Yaskawa INFORM job: DEMO_ROOF_SIDE_0625_3PAINT_8.JBI

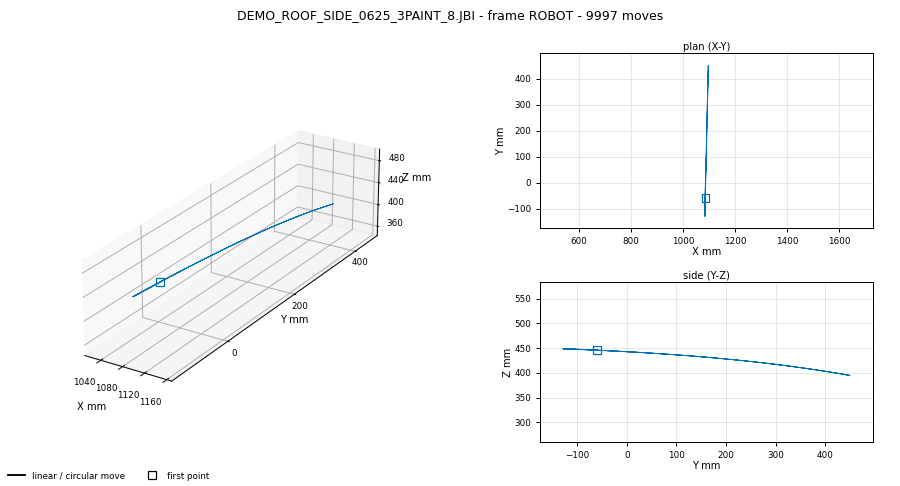
[picture p0: tool path of DEMO_ROOF_SIDE_0625_3PAINT_8.JBI in frame ROBOT, 9997 of 9997 moves have a stored position in this frame; points joined in program order, loops and branches not executed]
/JOB
//NAME DEMO_ROOF_SIDE_0625_3PAINT8
//POS
///NPOS 9997,0,0,0,0,0
///TOOL 0
///USER 0
///POSTYPE ROBOT
///RECTAN
///RCONF 1,0,0,0,0,0,0,0,0,0,0,0,0,0,0,0,0,0,0,0,0,0,0,0
C00000=1085.575,-60.075,446.143,174.285,17.982,152.948
C00001=1085.569,-60.325,446.155,174.283,17.980,152.948
C00002=1085.563,-60.574,446.167,174.282,17.979,152.948
C00003=1085.557,-60.824,446.178,174.280,17.978,152.948
C00004=1085.551,-61.074,446.189,174.279,17.976,152.948
C00005=1085.545,-61.323,446.201,174.277,17.974,152.948
C00006=1085.540,-61.573,446.212,174.276,17.973,152.948
C00007=1085.534,-61.823,446.223,174.274,17.972,152.948
C00008=1085.527,-62.072,446.235,174.273,17.970,152.948
C00009=1085.522,-62.322,446.246,174.272,17.969,152.948
C00010=1085.515,-62.572,446.257,174.270,17.968,152.948
C00011=1085.509,-62.821,446.269,174.269,17.966,152.948
C00012=1085.504,-63.071,446.281,174.267,17.965,152.948
C00013=1085.498,-63.321,446.292,174.265,17.963,152.948
C00014=1085.491,-63.571,446.303,174.264,17.962,152.948
C00015=1085.485,-63.820,446.315,174.263,17.960,152.948
C00016=1085.480,-64.069,446.325,174.261,17.959,152.948
C00017=1085.473,-64.320,446.337,174.260,17.958,152.948
C00018=1085.468,-64.569,446.349,174.258,17.956,152.948
C00019=1085.461,-64.842,446.360,174.257,17.955,152.948
C00020=1085.455,-65.116,446.373,174.254,17.953,152.948
C00021=1085.448,-65.389,446.385,174.253,17.951,152.948
C00022=1085.442,-65.662,446.398,174.252,17.950,152.948
C00023=1085.436,-65.912,446.409,174.250,17.948,152.948
C00024=1085.430,-66.162,446.420,174.248,17.947,152.948
C00025=1085.424,-66.411,446.431,174.247,17.946,152.948
C00026=1085.418,-66.661,446.443,174.246,17.944,152.948
C00027=1085.412,-66.911,446.454,174.244,17.943,152.948
C00028=1085.407,-67.160,446.465,174.243,17.942,152.948
C00029=1085.400,-67.410,446.476,174.241,17.940,152.948
C00030=1085.394,-67.660,446.487,174.240,17.939,152.948
C00031=1085.389,-67.909,446.498,174.238,17.937,152.948
C00032=1085.382,-68.159,446.510,174.237,17.936,152.948
C00033=1085.376,-68.409,446.521,174.235,17.935,152.948
C00034=1085.371,-68.658,446.532,174.234,17.933,152.948
C00035=1085.365,-68.909,446.544,174.232,17.932,152.948
C00036=1085.359,-69.158,446.555,174.231,17.931,152.948
C00037=1085.354,-69.407,446.565,174.229,17.929,152.948
C00038=1085.347,-69.658,446.577,174.228,17.928,152.948
C00039=1085.341,-69.907,446.588,174.226,17.926,152.948
C00040=1085.336,-70.157,446.598,174.225,17.925,152.948
C00041=1085.329,-70.406,446.610,174.223,17.924,152.948
C00042=1085.323,-70.656,446.621,174.222,17.922,152.948
C00043=1085.318,-70.905,446.632,174.220,17.921,152.948
C00044=1085.311,-71.155,446.643,174.219,17.920,152.948
C00045=1085.306,-71.405,446.654,174.217,17.918,152.948
C00046=1085.300,-71.655,446.666,174.216,17.917,152.948
C00047=1085.294,-71.905,446.677,174.214,17.915,152.948
C00048=1085.288,-72.154,446.688,174.213,17.914,152.948
C00049=1085.283,-72.404,446.699,174.211,17.913,152.949
C00050=1085.277,-72.653,446.710,174.210,17.911,152.948
C00051=1085.271,-72.904,446.721,174.208,17.910,152.948
C00052=1085.265,-73.153,446.732,174.207,17.909,152.949
C00053=1085.259,-73.403,446.743,174.205,17.907,152.949
C00054=1085.253,-73.652,446.754,174.204,17.906,152.949
C00055=1085.247,-73.902,446.765,174.202,17.904,152.949
C00056=1085.241,-74.152,446.776,174.201,17.903,152.949
C00057=1085.236,-74.401,446.787,174.199,17.902,152.949
C00058=1085.229,-74.651,446.798,174.198,17.900,152.949
C00059=1085.223,-74.901,446.809,174.196,17.899,152.949
C00060=1085.218,-75.150,446.820,174.195,17.898,152.949
C00061=1085.211,-75.400,446.830,174.193,17.896,152.949
C00062=1085.205,-75.650,446.841,174.192,17.895,152.949
C00063=1085.199,-75.899,446.852,174.190,17.894,152.949
C00064=1085.193,-76.149,446.863,174.188,17.893,152.949
C00065=1085.187,-76.399,446.874,174.187,17.891,152.949
C00066=1085.181,-76.648,446.885,174.185,17.890,152.949
C00067=1085.176,-76.898,446.896,174.184,17.889,152.949
C00068=1085.169,-77.148,446.906,174.182,17.888,152.949
C00069=1085.163,-77.398,446.917,174.181,17.886,152.949
C00070=1085.157,-77.647,446.927,174.179,17.885,152.949
C00071=1085.152,-77.897,446.938,174.178,17.883,152.949
C00072=1085.145,-78.147,446.950,174.176,17.882,152.949
C00073=1085.140,-78.397,446.960,174.175,17.881,152.949
C00074=1085.133,-78.646,446.971,174.174,17.880,152.949
C00075=1085.127,-78.895,446.982,174.172,17.879,152.949
C00076=1085.121,-79.145,446.993,174.171,17.878,152.949
C00077=1085.115,-79.395,447.004,174.169,17.876,152.949
C00078=1085.110,-79.645,447.014,174.168,17.875,152.949
C00079=1085.104,-79.894,447.025,174.166,17.874,152.950
C00080=1085.097,-80.144,447.035,174.165,17.872,152.950
C00081=1085.091,-80.394,447.046,174.163,17.871,152.950
C00082=1085.086,-80.643,447.057,174.162,17.870,152.950
C00083=1085.079,-80.920,447.069,174.160,17.869,152.950
C00084=1085.072,-81.195,447.081,174.158,17.868,152.950
C00085=1085.065,-81.470,447.093,174.157,17.866,152.950
C00086=1085.059,-81.746,447.104,174.154,17.865,152.950
C00087=1085.052,-81.995,447.114,174.153,17.863,152.950
C00088=1085.046,-82.245,447.126,174.152,17.862,152.950
C00089=1085.040,-82.495,447.136,174.150,17.861,152.950
C00090=1085.034,-82.744,447.146,174.149,17.860,152.950
C00091=1085.028,-82.994,447.157,174.147,17.859,152.950
C00092=1085.022,-83.244,447.168,174.146,17.858,152.950
C00093=1085.015,-83.493,447.178,174.144,17.857,152.950
C00094=1085.010,-83.743,447.189,174.143,17.855,152.950
C00095=1085.003,-83.993,447.199,174.141,17.854,152.950
C00096=1084.997,-84.243,447.210,174.139,17.853,152.951
C00097=1084.991,-84.492,447.221,174.138,17.851,152.951
C00098=1084.985,-84.742,447.231,174.136,17.850,152.951
C00099=1084.979,-84.992,447.241,174.135,17.849,152.951
C00100=1084.972,-85.241,447.252,174.133,17.848,152.951
C00101=1084.967,-85.492,447.262,174.132,17.847,152.951
C00102=1084.961,-85.741,447.273,174.131,17.846,152.951
C00103=1084.955,-85.990,447.283,174.129,17.845,152.951
C00104=1084.949,-86.240,447.294,174.128,17.844,152.951
C00105=1084.943,-86.491,447.305,174.126,17.842,152.951
C00106=1084.936,-86.740,447.315,174.124,17.841,152.951
C00107=1084.931,-86.990,447.325,174.123,17.840,152.951
C00108=1084.924,-87.239,447.335,174.121,17.839,152.951
C00109=1084.919,-87.488,447.346,174.120,17.838,152.951
C00110=1084.912,-87.739,447.356,174.118,17.836,152.951
C00111=1084.906,-87.988,447.367,174.117,17.835,152.952
C00112=1084.900,-88.238,447.378,174.115,17.834,152.952
C00113=1084.894,-88.488,447.388,174.114,17.834,152.952
C00114=1084.889,-88.737,447.398,174.113,17.832,152.952
C00115=1084.882,-88.986,447.409,174.111,17.831,152.952
C00116=1084.876,-89.237,447.419,174.109,17.830,152.952
C00117=1084.870,-89.486,447.430,174.108,17.829,152.952
C00118=1084.864,-89.737,447.440,174.106,17.827,152.952
C00119=1084.858,-89.986,447.451,174.105,17.826,152.952
C00120=1084.852,-90.235,447.461,174.103,17.825,152.952
C00121=1084.847,-90.485,447.471,174.101,17.824,152.952
C00122=1084.840,-90.734,447.481,174.101,17.823,152.952
C00123=1084.834,-90.985,447.492,174.099,17.822,152.952
C00124=1084.828,-91.234,447.502,174.097,17.821,152.952
C00125=1084.822,-91.485,447.512,174.096,17.820,152.953
C00126=1084.816,-91.734,447.523,174.094,17.819,152.953
C00127=1084.810,-91.984,447.533,174.093,17.817,152.953
C00128=1084.804,-92.233,447.543,174.091,17.816,152.953
C00129=1084.798,-92.483,447.554,174.089,17.815,152.953
C00130=1084.793,-92.733,447.564,174.088,17.814,152.953
C00131=1084.786,-92.982,447.574,174.087,17.813,152.953
C00132=1084.780,-93.233,447.585,174.085,17.812,152.953
C00133=1084.774,-93.482,447.595,174.084,17.811,152.953
C00134=1084.768,-93.732,447.605,174.082,17.810,152.953
C00135=1084.762,-93.981,447.616,174.080,17.809,152.953
C00136=1084.756,-94.231,447.626,174.079,17.807,152.953
C00137=1084.750,-94.480,447.636,174.077,17.806,152.953
C00138=1084.744,-94.731,447.646,174.076,17.805,152.954
C00139=1084.738,-94.980,447.656,174.074,17.804,152.954
C00140=1084.732,-95.230,447.667,174.073,17.804,152.954
C00141=1084.726,-95.480,447.676,174.072,17.803,152.954
C00142=1084.720,-95.729,447.687,174.070,17.801,152.954
C00143=1084.714,-95.979,447.697,174.068,17.800,152.954
C00144=1084.709,-96.228,447.708,174.067,17.799,152.954
C00145=1084.702,-96.478,447.717,174.065,17.798,152.954
C00146=1084.697,-96.728,447.727,174.063,17.797,152.954
C00147=1084.688,-97.066,447.741,174.062,17.796,152.954
C00148=1084.680,-97.404,447.755,174.060,17.794,152.954
C00149=1084.672,-97.741,447.769,174.058,17.793,152.954
C00150=1084.664,-98.079,447.782,174.055,17.791,152.955
C00151=1084.658,-98.328,447.793,174.054,17.790,152.955
C00152=1084.652,-98.578,447.802,174.053,17.789,152.955
C00153=1084.645,-98.828,447.812,174.051,17.788,152.955
C00154=1084.640,-99.077,447.823,174.050,17.787,152.955
C00155=1084.633,-99.328,447.833,174.048,17.786,152.955
C00156=1084.627,-99.577,447.842,174.046,17.785,152.955
C00157=1084.621,-99.827,447.853,174.045,17.784,152.955
C00158=1084.615,-100.077,447.863,174.044,17.784,152.955
C00159=1084.609,-100.326,447.872,174.042,17.783,152.956
C00160=1084.603,-100.576,447.883,174.040,17.782,152.956
C00161=1084.597,-100.826,447.893,174.039,17.781,152.956
C00162=1084.591,-101.076,447.902,174.037,17.779,152.956
C00163=1084.584,-101.325,447.912,174.035,17.778,152.956
C00164=1084.579,-101.575,447.923,174.035,17.778,152.956
C00165=1084.573,-101.825,447.932,174.033,17.777,152.956
C00166=1084.566,-102.074,447.942,174.031,17.776,152.956
C00167=1084.560,-102.324,447.952,174.030,17.775,152.956
C00168=1084.554,-102.574,447.962,174.028,17.774,152.957
C00169=1084.548,-102.824,447.972,174.026,17.773,152.957
C00170=1084.542,-103.073,447.982,174.026,17.772,152.957
C00171=1084.536,-103.323,447.992,174.024,17.771,152.957
C00172=1084.530,-103.573,448.002,174.022,17.770,152.957
C00173=1084.524,-103.822,448.011,174.021,17.769,152.957
C00174=1084.518,-104.072,448.022,174.019,17.768,152.957
C00175=1084.512,-104.322,448.032,174.017,17.767,152.957
C00176=1084.506,-104.571,448.041,174.016,17.766,152.957
C00177=1084.500,-104.821,448.051,174.015,17.765,152.957
C00178=1084.493,-105.070,448.061,174.013,17.764,152.958
C00179=1084.487,-105.320,448.071,174.011,17.763,152.958
C00180=1084.482,-105.570,448.081,174.010,17.762,152.958
C00181=1084.475,-105.820,448.090,174.009,17.762,152.958
C00182=1084.469,-106.070,448.100,174.007,17.761,152.958
C00183=1084.463,-106.319,448.110,174.006,17.760,152.958
C00184=1084.457,-106.569,448.120,174.004,17.758,152.958
C00185=1084.451,-106.819,448.130,174.002,17.758,152.958
C00186=1084.445,-107.069,448.140,174.000,17.757,152.959
C00187=1084.439,-107.319,448.149,173.999,17.756,152.959
C00188=1084.433,-107.568,448.159,173.998,17.755,152.959
C00189=1084.426,-107.818,448.169,173.996,17.754,152.959
C00190=1084.420,-108.067,448.179,173.994,17.753,152.959
C00191=1084.414,-108.317,448.188,173.993,17.752,152.959
C00192=1084.408,-108.567,448.198,173.992,17.752,152.959
C00193=1084.402,-108.817,448.208,173.990,17.751,152.959
C00194=1084.396,-109.067,448.217,173.988,17.750,152.960
C00195=1084.390,-109.317,448.227,173.987,17.749,152.960
C00196=1084.384,-109.567,448.237,173.985,17.748,152.960
C00197=1084.377,-109.816,448.247,173.984,17.747,152.960
C00198=1084.371,-110.065,448.256,173.983,17.746,152.960
C00199=1084.365,-110.315,448.266,173.981,17.746,152.960
C00200=1084.359,-110.565,448.276,173.979,17.745,152.960
C00201=1084.353,-110.815,448.285,173.978,17.744,152.960
C00202=1084.347,-111.064,448.294,173.976,17.743,152.961
C00203=1084.342,-111.284,448.303,173.975,17.742,152.961
C00204=1084.336,-111.504,448.312,173.974,17.742,152.961
C00205=1084.331,-111.724,448.320,173.972,17.741,152.961
C00206=1084.325,-111.944,448.329,173.970,17.740,152.961
C00207=1084.321,-112.163,448.337,173.970,17.740,152.961
C00208=1084.315,-112.383,448.346,173.968,17.739,152.961
C00209=1084.310,-112.604,448.354,173.967,17.738,152.961
C00210=1084.304,-112.823,448.362,173.965,17.737,152.962
C00211=1084.298,-113.096,448.373,173.963,17.736,152.962
C00212=1084.291,-113.370,448.384,173.962,17.735,152.962
C00213=1084.284,-113.643,448.394,173.960,17.734,152.962
C00214=1084.277,-113.917,448.405,173.958,17.734,152.962
C00215=1084.271,-114.167,448.414,173.957,17.733,152.962
C00216=1084.265,-114.417,448.424,173.956,17.732,152.962
C00217=1084.259,-114.667,448.433,173.954,17.731,152.963
C00218=1084.253,-114.916,448.443,173.952,17.731,152.963
C00219=1084.247,-115.166,448.452,173.951,17.730,152.963
C00220=1084.241,-115.416,448.461,173.950,17.729,152.963
C00221=1084.235,-115.666,448.471,173.948,17.729,152.963
C00222=1084.229,-115.916,448.480,173.946,17.727,152.963
C00223=1084.223,-116.165,448.490,173.945,17.727,152.963
C00224=1084.217,-116.415,448.499,173.943,17.726,152.964
C00225=1084.210,-116.665,448.509,173.942,17.725,152.964
C00226=1084.203,-116.914,448.518,173.940,17.724,152.964
C00227=1084.197,-117.164,448.527,173.939,17.724,152.964
C00228=1084.191,-117.414,448.537,173.937,17.723,152.964
C00229=1084.186,-117.663,448.546,173.936,17.722,152.964
C00230=1084.179,-117.913,448.556,173.934,17.721,152.964
C00231=1084.173,-118.163,448.565,173.933,17.721,152.965
C00232=1084.167,-118.412,448.575,173.931,17.720,152.965
C00233=1084.161,-118.663,448.584,173.929,17.720,152.965
C00234=1084.155,-118.913,448.593,173.927,17.719,152.965
C00235=1084.149,-119.163,448.603,173.927,17.718,152.965
C00236=1084.143,-119.412,448.612,173.925,17.718,152.965
C00237=1084.136,-119.661,448.621,173.923,17.716,152.966
C00238=1084.130,-119.911,448.631,173.921,17.715,152.966
C00239=1084.124,-120.161,448.640,173.920,17.715,152.966
C00240=1084.118,-120.410,448.650,173.919,17.714,152.966
C00241=1084.112,-120.661,448.659,173.917,17.714,152.966
C00242=1084.106,-120.911,448.668,173.915,17.713,152.966
C00243=1084.100,-121.160,448.677,173.914,17.712,152.966
C00244=1084.094,-121.410,448.687,173.912,17.712,152.967
C00245=1084.087,-121.659,448.696,173.911,17.711,152.967
C00246=1084.081,-121.910,448.705,173.910,17.711,152.967
C00247=1084.075,-122.159,448.714,173.908,17.710,152.967
C00248=1084.069,-122.409,448.724,173.906,17.709,152.967
C00249=1084.063,-122.658,448.733,173.904,17.708,152.968
C00250=1084.057,-122.908,448.743,173.903,17.708,152.968
C00251=1084.051,-123.158,448.751,173.901,17.707,152.968
C00252=1084.044,-123.408,448.760,173.900,17.706,152.968
C00253=1084.038,-123.658,448.770,173.899,17.706,152.968
C00254=1084.032,-123.907,448.780,173.897,17.705,152.968
C00255=1084.027,-124.157,448.789,173.895,17.704,152.969
C00256=1084.020,-124.407,448.797,173.893,17.703,152.969
C00257=1084.014,-124.656,448.807,173.892,17.703,152.969
C00258=1084.008,-124.906,448.816,173.891,17.702,152.969
C00259=1084.002,-125.157,448.825,173.889,17.702,152.969
C00260=1083.995,-125.405,448.834,173.888,17.701,152.969
C00261=1083.989,-125.655,448.843,173.886,17.701,152.970
C00262=1083.983,-125.905,448.853,173.884,17.700,152.970
C00263=1083.977,-126.156,448.862,173.882,17.699,152.970
C00264=1083.970,-126.405,448.871,173.882,17.699,152.970
C00265=1083.965,-126.654,448.880,173.880,17.698,152.970
C00266=1083.959,-126.905,448.889,173.878,17.697,152.970
C00267=1083.953,-127.154,448.898,173.877,17.697,152.971
C00268=1083.946,-127.404,448.907,173.875,17.696,152.971
C00269=1083.940,-127.654,448.917,173.873,17.695,152.971
C00270=1083.934,-127.903,448.925,173.872,17.695,152.971
C00271=1083.928,-128.160,448.935,173.871,17.694,152.971
C00272=1083.927,-128.416,448.946,173.869,17.692,152.971
C00273=1083.930,-128.671,448.958,173.869,17.689,152.971
C00274=1083.937,-128.924,448.972,173.869,17.684,152.970
C00275=1083.537,-128.945,448.838,173.825,17.800,153.000
C00276=1083.528,-128.693,448.824,173.825,17.805,153.001
C00277=1083.525,-128.438,448.812,173.826,17.808,153.001
C00278=1083.527,-128.182,448.801,173.827,17.810,153.001
C00279=1083.532,-127.926,448.791,173.828,17.811,153.001
C00280=1083.538,-127.676,448.782,173.829,17.812,153.001
C00281=1083.544,-127.426,448.773,173.831,17.812,153.001
C00282=1083.550,-127.176,448.763,173.833,17.813,153.001
C00283=1083.556,-126.927,448.755,173.835,17.814,153.001
C00284=1083.563,-126.677,448.745,173.836,17.814,153.001
C00285=1083.568,-126.427,448.736,173.838,17.815,153.000
C00286=1083.575,-126.177,448.727,173.839,17.816,153.000
C00287=1083.582,-125.927,448.718,173.840,17.816,153.000
C00288=1083.587,-125.678,448.709,173.842,17.817,153.000
C00289=1083.593,-125.428,448.700,173.844,17.817,153.000
C00290=1083.600,-125.178,448.691,173.846,17.819,152.999
C00291=1083.606,-124.929,448.681,173.847,17.819,152.999
C00292=1083.612,-124.678,448.672,173.848,17.820,152.999
C00293=1083.617,-124.429,448.663,173.850,17.820,152.999
C00294=1083.624,-124.180,448.654,173.851,17.821,152.999
C00295=1083.631,-123.930,448.645,173.853,17.821,152.999
C00296=1083.636,-123.679,448.636,173.855,17.822,152.998
C00297=1083.643,-123.430,448.626,173.857,17.823,152.998
C00298=1083.649,-123.180,448.617,173.858,17.823,152.998
C00299=1083.654,-122.931,448.607,173.859,17.824,152.998
C00300=1083.661,-122.681,448.599,173.861,17.825,152.998
C00301=1083.667,-122.431,448.590,173.862,17.825,152.998
C00302=1083.673,-122.181,448.580,173.864,17.826,152.997
C00303=1083.679,-121.931,448.571,173.866,17.827,152.997
C00304=1083.685,-121.682,448.561,173.867,17.828,152.997
C00305=1083.691,-121.432,448.552,173.868,17.828,152.997
C00306=1083.698,-121.182,448.543,173.870,17.829,152.997
C00307=1083.704,-120.932,448.534,173.872,17.829,152.997
C00308=1083.710,-120.683,448.524,173.874,17.830,152.996
C00309=1083.716,-120.433,448.515,173.874,17.831,152.996
C00310=1083.722,-120.183,448.505,173.876,17.832,152.996
C00311=1083.728,-119.933,448.497,173.878,17.833,152.996
C00312=1083.734,-119.684,448.487,173.880,17.834,152.996
C00313=1083.741,-119.434,448.478,173.881,17.834,152.996
C00314=1083.747,-119.184,448.469,173.882,17.835,152.996
C00315=1083.753,-118.934,448.459,173.884,17.836,152.995
C00316=1083.759,-118.685,448.449,173.886,17.836,152.995
C00317=1083.766,-118.435,448.440,173.887,17.837,152.995
C00318=1083.771,-118.186,448.431,173.889,17.838,152.995
C00319=1083.777,-117.935,448.422,173.891,17.838,152.995
C00320=1083.783,-117.686,448.412,173.892,17.839,152.995
C00321=1083.789,-117.436,448.403,173.893,17.840,152.995
C00322=1083.795,-117.186,448.393,173.895,17.840,152.994
C00323=1083.802,-116.936,448.384,173.897,17.841,152.994
C00324=1083.808,-116.686,448.374,173.898,17.842,152.994
C00325=1083.815,-116.437,448.365,173.899,17.842,152.994
C00326=1083.821,-116.187,448.355,173.901,17.844,152.994
C00327=1083.826,-115.938,448.346,173.903,17.845,152.994
C00328=1083.833,-115.688,448.337,173.904,17.846,152.993
C00329=1083.839,-115.438,448.327,173.905,17.846,152.993
C00330=1083.845,-115.189,448.318,173.907,17.847,152.993
C00331=1083.851,-114.939,448.308,173.909,17.848,152.993
C00332=1083.857,-114.689,448.298,173.910,17.849,152.993
C00333=1083.864,-114.439,448.289,173.912,17.849,152.993
C00334=1083.870,-114.189,448.279,173.913,17.850,152.993
C00335=1083.876,-113.940,448.270,173.915,17.851,152.992
C00336=1083.882,-113.666,448.260,173.917,17.852,152.992
C00337=1083.888,-113.392,448.249,173.918,17.853,152.992
C00338=1083.895,-113.118,448.238,173.920,17.853,152.992
C00339=1083.903,-112.844,448.228,173.922,17.854,152.992
C00340=1083.909,-112.595,448.218,173.924,17.856,152.992
C00341=1083.915,-112.345,448.209,173.924,17.856,152.992
C00342=1083.921,-112.095,448.199,173.926,17.857,152.992
C00343=1083.927,-111.846,448.190,173.928,17.858,152.991
C00344=1083.932,-111.596,448.180,173.930,17.859,152.991
C00345=1083.938,-111.346,448.170,173.931,17.860,152.991
C00346=1083.944,-111.096,448.161,173.932,17.860,152.991
C00347=1083.951,-110.846,448.151,173.934,17.861,152.991
C00348=1083.957,-110.597,448.141,173.935,17.862,152.991
C00349=1083.963,-110.347,448.132,173.937,17.863,152.990
C00350=1083.969,-110.097,448.122,173.939,17.864,152.990
C00351=1083.975,-109.847,448.113,173.940,17.864,152.990
C00352=1083.982,-109.597,448.103,173.942,17.865,152.990
C00353=1083.988,-109.348,448.094,173.943,17.866,152.990
C00354=1083.994,-109.098,448.083,173.945,17.868,152.990
C00355=1084.000,-108.849,448.074,173.947,17.869,152.990
C00356=1084.007,-108.599,448.064,173.948,17.869,152.990
C00357=1084.012,-108.349,448.054,173.949,17.870,152.990
C00358=1084.018,-108.099,448.044,173.951,17.871,152.989
C00359=1084.024,-107.849,448.035,173.953,17.872,152.989
C00360=1084.030,-107.599,448.025,173.954,17.873,152.989
C00361=1084.037,-107.350,448.015,173.955,17.873,152.989
C00362=1084.043,-107.100,448.005,173.957,17.874,152.989
C00363=1084.049,-106.850,447.996,173.958,17.875,152.989
C00364=1084.055,-106.600,447.986,173.960,17.876,152.989
C00365=1084.061,-106.351,447.976,173.962,17.877,152.989
C00366=1084.067,-106.101,447.967,173.963,17.878,152.989
C00367=1084.074,-105.852,447.956,173.964,17.879,152.988
C00368=1084.080,-105.602,447.947,173.966,17.880,152.988
C00369=1084.085,-105.352,447.937,173.968,17.881,152.988
C00370=1084.091,-105.102,447.927,173.969,17.882,152.988
C00371=1084.097,-104.852,447.917,173.971,17.883,152.988
C00372=1084.104,-104.603,447.907,173.972,17.883,152.988
C00373=1084.109,-104.353,447.897,173.974,17.884,152.988
C00374=1084.116,-104.103,447.887,173.975,17.885,152.988
C00375=1084.122,-103.853,447.878,173.977,17.886,152.987
C00376=1084.128,-103.604,447.868,173.979,17.887,152.987
C00377=1084.134,-103.354,447.857,173.980,17.888,152.987
C00378=1084.140,-103.104,447.848,173.981,17.889,152.987
C00379=1084.146,-102.854,447.838,173.983,17.890,152.987
C00380=1084.152,-102.605,447.828,173.984,17.892,152.987
C00381=1084.158,-102.355,447.818,173.986,17.893,152.987
C00382=1084.164,-102.105,447.808,173.988,17.894,152.987
C00383=1084.170,-101.855,447.799,173.989,17.895,152.987
C00384=1084.177,-101.606,447.788,173.990,17.895,152.987
C00385=1084.182,-101.356,447.778,173.992,17.896,152.987
C00386=1084.188,-101.106,447.769,173.993,17.897,152.986
C00387=1084.195,-100.857,447.758,173.995,17.898,152.986
C00388=1084.200,-100.607,447.748,173.997,17.899,152.986
C00389=1084.206,-100.357,447.739,173.998,17.900,152.986
C00390=1084.213,-100.108,447.728,173.999,17.901,152.986
C00391=1084.219,-99.858,447.719,174.001,17.902,152.986
C00392=1084.224,-99.608,447.709,174.003,17.903,152.986
C00393=1084.231,-99.359,447.698,174.004,17.904,152.986
C00394=1084.237,-99.109,447.689,174.006,17.905,152.986
C00395=1084.243,-98.859,447.679,174.008,17.906,152.985
C00396=1084.249,-98.610,447.668,174.009,17.907,152.985
C00397=1084.255,-98.360,447.659,174.010,17.908,152.985
C00398=1084.262,-98.110,447.648,174.012,17.909,152.985
C00399=1084.268,-97.860,447.638,174.013,17.910,152.985
C00400=1084.275,-97.582,447.627,174.015,17.911,152.985
C00401=1084.281,-97.304,447.616,174.017,17.912,152.985
C00402=1084.288,-97.026,447.605,174.018,17.913,152.985
C00403=1084.295,-96.748,447.593,174.020,17.914,152.985
C00404=1084.300,-96.498,447.583,174.021,17.916,152.985
C00405=1084.307,-96.249,447.572,174.023,17.917,152.985
C00406=1084.313,-95.999,447.563,174.025,17.918,152.985
C00407=1084.318,-95.750,447.552,174.026,17.919,152.984
C00408=1084.325,-95.500,447.542,174.028,17.920,152.984
C00409=1084.330,-95.250,447.532,174.029,17.922,152.984
C00410=1084.337,-95.001,447.522,174.031,17.923,152.984
C00411=1084.342,-94.751,447.512,174.032,17.923,152.984
C00412=1084.348,-94.501,447.502,174.034,17.924,152.984
C00413=1084.354,-94.251,447.491,174.035,17.926,152.984
C00414=1084.360,-94.002,447.481,174.037,17.927,152.984
C00415=1084.366,-93.752,447.471,174.038,17.928,152.984
C00416=1084.372,-93.503,447.460,174.040,17.929,152.984
C00417=1084.378,-93.253,447.450,174.042,17.930,152.984
C00418=1084.384,-93.003,447.439,174.043,17.932,152.984
C00419=1084.390,-92.753,447.430,174.044,17.932,152.984
C00420=1084.396,-92.503,447.419,174.045,17.933,152.984
C00421=1084.402,-92.253,447.409,174.047,17.934,152.983
C00422=1084.408,-92.004,447.398,174.049,17.936,152.983
C00423=1084.414,-91.754,447.389,174.050,17.937,152.983
C00424=1084.420,-91.505,447.378,174.052,17.938,152.983
C00425=1084.426,-91.255,447.368,174.054,17.939,152.983
C00426=1084.432,-91.005,447.357,174.055,17.941,152.983
C00427=1084.439,-90.756,447.347,174.057,17.942,152.983
C00428=1084.444,-90.505,447.337,174.058,17.943,152.983
C00429=1084.451,-90.256,447.326,174.059,17.944,152.983
C00430=1084.456,-90.006,447.316,174.061,17.945,152.983
C00431=1084.462,-89.757,447.305,174.062,17.946,152.983
C00432=1084.468,-89.507,447.295,174.064,17.947,152.983
C00433=1084.474,-89.257,447.285,174.065,17.948,152.983
C00434=1084.481,-89.007,447.274,174.067,17.949,152.983
C00435=1084.486,-88.757,447.264,174.069,17.951,152.982
C00436=1084.493,-88.508,447.254,174.070,17.952,152.982
C00437=1084.499,-88.259,447.243,174.072,17.953,152.982
C00438=1084.504,-88.009,447.233,174.073,17.954,152.982
C00439=1084.510,-87.759,447.222,174.074,17.955,152.982
C00440=1084.517,-87.509,447.211,174.076,17.956,152.982
C00441=1084.523,-87.259,447.202,174.077,17.957,152.982
C00442=1084.529,-87.010,447.191,174.079,17.959,152.982
C00443=1084.534,-86.760,447.180,174.080,17.960,152.982
C00444=1084.541,-86.511,447.170,174.082,17.961,152.982
C00445=1084.547,-86.260,447.159,174.084,17.962,152.982
C00446=1084.553,-86.011,447.149,174.085,17.964,152.982
C00447=1084.559,-85.761,447.139,174.087,17.965,152.982
C00448=1084.565,-85.512,447.128,174.088,17.966,152.982
C00449=1084.571,-85.262,447.117,174.090,17.967,152.982
C00450=1084.577,-85.012,447.107,174.091,17.968,152.982
C00451=1084.584,-84.762,447.097,174.092,17.969,152.982
C00452=1084.589,-84.513,447.086,174.094,17.970,152.982
C00453=1084.595,-84.264,447.075,174.095,17.971,152.981
C00454=1084.602,-84.013,447.065,174.097,17.973,152.981
C00455=1084.608,-83.764,447.054,174.098,17.974,152.981
C00456=1084.614,-83.514,447.044,174.100,17.975,152.981
C00457=1084.620,-83.265,447.033,174.102,17.977,152.981
C00458=1084.626,-83.014,447.022,174.103,17.978,152.981
C00459=1084.632,-82.765,447.012,174.105,17.979,152.981
C00460=1084.638,-82.515,447.001,174.106,17.980,152.981
C00461=1084.644,-82.266,446.990,174.108,17.981,152.981
C00462=1084.651,-82.016,446.980,174.109,17.983,152.981
C00463=1084.656,-81.766,446.970,174.111,17.984,152.981
C00464=1084.663,-81.491,446.958,174.113,17.985,152.981
C00465=1084.670,-81.215,446.946,174.114,17.987,152.981
C00466=1084.677,-80.939,446.934,174.116,17.988,152.981
C00467=1084.683,-80.663,446.923,174.117,17.989,152.981
C00468=1084.689,-80.414,446.912,174.119,17.990,152.981
C00469=1084.696,-80.164,446.901,174.120,17.991,152.981
C00470=1084.702,-79.915,446.890,174.122,17.993,152.981
C00471=1084.708,-79.665,446.879,174.124,17.994,152.980
C00472=1084.714,-79.415,446.868,174.125,17.995,152.980
C00473=1084.719,-79.165,446.858,174.127,17.996,152.980
C00474=1084.726,-78.916,446.848,174.128,17.998,152.980
C00475=1084.732,-78.666,446.837,174.130,17.999,152.980
C00476=1084.738,-78.416,446.826,174.131,18.001,152.980
C00477=1084.744,-78.166,446.815,174.133,18.002,152.980
C00478=1084.749,-77.917,446.804,174.134,18.003,152.980
C00479=1084.755,-77.667,446.793,174.136,18.004,152.980
C00480=1084.761,-77.417,446.782,174.137,18.006,152.980
C00481=1084.768,-77.168,446.772,174.139,18.007,152.980
C00482=1084.773,-76.918,446.761,174.140,18.008,152.980
C00483=1084.779,-76.668,446.750,174.142,18.010,152.980
C00484=1084.785,-76.418,446.739,174.143,18.011,152.980
C00485=1084.791,-76.169,446.728,174.145,18.013,152.980
C00486=1084.797,-75.919,446.717,174.146,18.014,152.980
C00487=1084.803,-75.669,446.706,174.147,18.015,152.980
C00488=1084.810,-75.420,446.696,174.149,18.016,152.980
C00489=1084.815,-75.170,446.685,174.150,18.017,152.980
C00490=1084.822,-74.920,446.674,174.152,18.018,152.980
C00491=1084.828,-74.671,446.663,174.153,18.020,152.980
C00492=1084.833,-74.421,446.652,174.155,18.021,152.980
C00493=1084.839,-74.172,446.641,174.156,18.023,152.980
C00494=1084.845,-73.922,446.630,174.158,18.024,152.980
C00495=1084.851,-73.672,446.619,174.159,18.025,152.980
C00496=1084.857,-73.423,446.608,174.161,18.027,152.980
C00497=1084.863,-73.172,446.597,174.162,18.028,152.980
C00498=1084.869,-72.923,446.586,174.164,18.029,152.980
C00499=1084.875,-72.673,446.575,174.165,18.031,152.980
C00500=1084.880,-72.424,446.564,174.167,18.032,152.980
C00501=1084.887,-72.174,446.553,174.168,18.033,152.980
C00502=1084.892,-71.924,446.542,174.170,18.035,152.980
C00503=1084.898,-71.675,446.531,174.171,18.036,152.980
C00504=1084.905,-71.425,446.520,174.173,18.038,152.980
C00505=1084.910,-71.175,446.509,174.174,18.039,152.980
C00506=1084.915,-70.925,446.498,174.176,18.040,152.980
C00507=1084.921,-70.676,446.486,174.177,18.042,152.980
C00508=1084.928,-70.426,446.475,174.179,18.043,152.980
C00509=1084.933,-70.177,446.464,174.180,18.044,152.979
C00510=1084.939,-69.927,446.453,174.182,18.046,152.980
C00511=1084.946,-69.677,446.442,174.183,18.048,152.980
C00512=1084.951,-69.428,446.431,174.184,18.049,152.980
C00513=1084.957,-69.178,446.420,174.186,18.050,152.979
C00514=1084.963,-68.928,446.409,174.188,18.052,152.980
C00515=1084.969,-68.678,446.398,174.189,18.053,152.980
C00516=1084.975,-68.430,446.386,174.191,18.054,152.979
C00517=1084.981,-68.179,446.375,174.192,18.056,152.979
C00518=1084.986,-67.930,446.364,174.193,18.057,152.980
C00519=1084.992,-67.680,446.353,174.195,18.059,152.979
C00520=1084.999,-67.430,446.342,174.197,18.060,152.979
C00521=1085.004,-67.180,446.331,174.198,18.062,152.979
C00522=1085.010,-66.932,446.319,174.199,18.063,152.980
C00523=1085.017,-66.681,446.308,174.201,18.064,152.979
C00524=1085.022,-66.432,446.297,174.202,18.066,152.979
C00525=1085.028,-66.181,446.285,174.204,18.067,152.979
C00526=1085.034,-65.932,446.274,174.205,18.068,152.979
C00527=1085.040,-65.683,446.263,174.207,18.070,152.979
C00528=1085.046,-65.409,446.250,174.209,18.072,152.979
C00529=1085.053,-65.135,446.238,174.211,18.074,152.979
C00530=1085.059,-64.861,446.226,174.212,18.075,152.979
C00531=1085.066,-64.588,446.214,174.214,18.076,152.979
C00532=1085.072,-64.339,446.202,174.215,18.078,152.979
C00533=1085.078,-64.089,446.191,174.216,18.079,152.979
C00534=1085.084,-63.839,446.180,174.218,18.081,152.979
C00535=1085.089,-63.590,446.169,174.219,18.082,152.979
C00536=1085.096,-63.340,446.157,174.221,18.084,152.979
C00537=1085.102,-63.091,446.146,174.222,18.085,152.979
C00538=1085.107,-62.840,446.134,174.225,18.087,152.979
C00539=1085.114,-62.591,446.123,174.226,18.088,152.979
C00540=1085.120,-62.341,446.111,174.228,18.090,152.979
C00541=1085.126,-62.092,446.100,174.229,18.091,152.979
C00542=1085.132,-61.843,446.089,174.230,18.093,152.979
C00543=1085.137,-61.592,446.077,174.232,18.094,152.979
C00544=1085.143,-61.343,446.066,174.233,18.096,152.979
C00545=1085.150,-61.093,446.054,174.235,18.097,152.979
C00546=1085.155,-60.844,446.043,174.236,18.099,152.979
C00547=1085.162,-60.594,446.032,174.238,18.100,152.979
C00548=1085.167,-60.344,446.020,174.239,18.101,152.979
C00549=1085.173,-60.094,446.009,174.241,18.103,152.979
C00550=1085.179,-59.845,445.998,174.242,18.104,152.979
C00551=1085.186,-59.595,445.986,174.244,18.105,152.979
C00552=1085.191,-59.346,445.975,174.245,18.107,152.979
C00553=1085.197,-59.096,445.962,174.247,18.109,152.979
C00554=1085.203,-58.846,445.951,174.248,18.110,152.979
C00555=1085.209,-58.596,445.940,174.249,18.112,152.979
C00556=1085.216,-58.347,445.929,174.251,18.113,152.979
C00557=1085.221,-58.097,445.917,174.253,18.114,152.979
C00558=1085.227,-57.848,445.905,174.254,18.116,152.979
C00559=1085.233,-57.598,445.894,174.255,18.117,152.979
C00560=1085.240,-57.349,445.882,174.257,18.119,152.980
C00561=1085.246,-57.099,445.871,174.259,18.120,152.979
C00562=1085.251,-56.849,445.860,174.261,18.122,152.979
C00563=1085.258,-56.599,445.848,174.262,18.124,152.979
C00564=1085.263,-56.350,445.837,174.264,18.125,152.979
C00565=1085.269,-56.100,445.824,174.265,18.127,152.980
C00566=1085.276,-55.850,445.813,174.267,18.128,152.979
C00567=1085.282,-55.601,445.801,174.268,18.129,152.979
C00568=1085.288,-55.351,445.790,174.269,18.131,152.979
C00569=1085.293,-55.101,445.778,174.271,18.132,152.980
C00570=1085.300,-54.851,445.767,174.272,18.134,152.980
C00571=1085.306,-54.602,445.755,174.274,18.135,152.979
C00572=1085.312,-54.352,445.744,174.275,18.137,152.979
C00573=1085.318,-54.102,445.731,174.277,18.138,152.980
C00574=1085.324,-53.853,445.720,174.278,18.140,152.980
C00575=1085.330,-53.603,445.709,174.280,18.141,152.980
C00576=1085.336,-53.354,445.696,174.281,18.142,152.979
C00577=1085.342,-53.104,445.685,174.283,18.144,152.979
C00578=1085.349,-52.854,445.673,174.285,18.146,152.980
C00579=1085.354,-52.605,445.662,174.286,18.148,152.980
C00580=1085.360,-52.355,445.650,174.288,18.149,152.980
C00581=1085.366,-52.106,445.638,174.289,18.151,152.980
C00582=1085.373,-51.856,445.627,174.291,18.152,152.980
C00583=1085.378,-51.606,445.614,174.292,18.153,152.980
C00584=1085.384,-51.356,445.603,174.294,18.155,152.980
C00585=1085.391,-51.107,445.591,174.295,18.156,152.980
C00586=1085.397,-50.857,445.579,174.296,18.158,152.980
C00587=1085.402,-50.607,445.568,174.298,18.160,152.980
C00588=1085.409,-50.358,445.556,174.299,18.161,152.980
C00589=1085.414,-50.108,445.545,174.301,18.162,152.980
C00590=1085.421,-49.859,445.533,174.303,18.164,152.980
C00591=1085.426,-49.609,445.520,174.304,18.166,152.980
C00592=1085.433,-49.336,445.508,174.306,18.167,152.980
C00593=1085.439,-49.065,445.494,174.307,18.169,152.980
C00594=1085.445,-48.792,445.482,174.310,18.171,152.980
C00595=1085.452,-48.520,445.468,174.311,18.173,152.980
C00596=1085.458,-48.271,445.457,174.312,18.174,152.980
C00597=1085.464,-48.021,445.445,174.314,18.176,152.980
C00598=1085.470,-47.772,445.433,174.315,18.177,152.980
C00599=1085.475,-47.521,445.421,174.317,18.179,152.980
C00600=1085.482,-47.272,445.409,174.318,18.180,152.980
C00601=1085.487,-47.023,445.397,174.319,18.182,152.980
C00602=1085.493,-46.773,445.384,174.321,18.183,152.980
C00603=1085.499,-46.523,445.374,174.323,18.186,152.980
C00604=1085.505,-46.273,445.361,174.324,18.187,152.980
C00605=1085.511,-46.024,445.349,174.326,18.189,152.980
C00606=1085.517,-45.775,445.337,174.327,18.190,152.980
C00607=1085.522,-45.524,445.325,174.329,18.192,152.980
C00608=1085.532,-45.122,445.306,174.331,18.194,152.980
C00609=1085.541,-44.720,445.286,174.334,18.197,152.980
C00610=1085.551,-44.318,445.267,174.336,18.200,152.980
C00611=1085.560,-43.916,445.247,174.339,18.203,152.980
C00612=1085.567,-43.666,445.235,174.340,18.204,152.981
C00613=1085.573,-43.416,445.223,174.341,18.206,152.981
C00614=1085.579,-43.167,445.212,174.343,18.207,152.981
C00615=1085.584,-42.917,445.199,174.344,18.209,152.981
C00616=1085.590,-42.667,445.187,174.346,18.210,152.981
C00617=1085.596,-42.418,445.175,174.347,18.212,152.981
C00618=1085.602,-42.168,445.163,174.348,18.214,152.981
C00619=1085.608,-41.918,445.150,174.351,18.216,152.981
C00620=1085.615,-41.669,445.138,174.352,18.217,152.981
C00621=1085.620,-41.419,445.127,174.353,18.219,152.981
C00622=1085.626,-41.169,445.114,174.355,18.220,152.981
C00623=1085.632,-40.920,445.102,174.356,18.222,152.981
C00624=1085.638,-40.670,445.090,174.358,18.223,152.981
C00625=1085.644,-40.420,445.077,174.359,18.225,152.981
C00626=1085.650,-40.171,445.066,174.361,18.227,152.981
C00627=1085.656,-39.922,445.053,174.363,18.229,152.981
C00628=1085.662,-39.672,445.041,174.364,18.230,152.981
C00629=1085.668,-39.422,445.029,174.366,18.232,152.981
C00630=1085.674,-39.172,445.016,174.367,18.233,152.981
C00631=1085.679,-38.923,445.004,174.368,18.235,152.981
C00632=1085.686,-38.674,444.992,174.370,18.236,152.981
C00633=1085.692,-38.424,444.980,174.371,18.238,152.981
C00634=1085.698,-38.173,444.968,174.373,18.240,152.981
C00635=1085.703,-37.924,444.956,174.375,18.242,152.981
C00636=1085.709,-37.674,444.943,174.376,18.243,152.981
C00637=1085.715,-37.425,444.931,174.378,18.245,152.981
C00638=1085.721,-37.175,444.919,174.379,18.246,152.981
C00639=1085.727,-36.926,444.906,174.381,18.248,152.981
C00640=1085.733,-36.676,444.894,174.382,18.249,152.981
C00641=1085.738,-36.426,444.882,174.383,18.251,152.982
C00642=1085.744,-36.177,444.869,174.385,18.254,152.982
C00643=1085.750,-35.927,444.857,174.387,18.255,152.982
C00644=1085.757,-35.678,444.844,174.388,18.257,152.982
C00645=1085.762,-35.429,444.832,174.390,18.258,152.982
C00646=1085.768,-35.179,444.819,174.391,18.260,152.982
C00647=1085.774,-34.929,444.806,174.392,18.261,152.982
C00648=1085.780,-34.679,444.794,174.394,18.263,152.982
C00649=1085.785,-34.430,444.782,174.396,18.265,152.982
C00650=1085.791,-34.180,444.769,174.397,18.267,152.982
C00651=1085.797,-33.930,444.757,174.399,18.269,152.982
C00652=1085.806,-33.561,444.739,174.401,18.271,152.982
C00653=1085.815,-33.193,444.720,174.403,18.273,152.982
C00654=1085.823,-32.824,444.702,174.405,18.275,152.982
C00655=1085.832,-32.455,444.683,174.408,18.278,152.982
C00656=1085.838,-32.205,444.671,174.409,18.280,152.982
C00657=1085.844,-31.956,444.659,174.411,18.282,152.982
C00658=1085.849,-31.706,444.646,174.412,18.283,152.982
C00659=1085.855,-31.456,444.633,174.413,18.285,152.983
C00660=1085.861,-31.206,444.621,174.415,18.287,152.983
C00661=1085.868,-30.957,444.608,174.417,18.289,152.983
C00662=1085.873,-30.708,444.595,174.418,18.290,152.983
C00663=1085.879,-30.458,444.583,174.420,18.292,152.983
C00664=1085.885,-30.208,444.570,174.421,18.294,152.983
C00665=1085.891,-29.958,444.558,174.423,18.295,152.983
C00666=1085.897,-29.709,444.544,174.424,18.297,152.983
C00667=1085.903,-29.459,444.532,174.426,18.299,152.983
C00668=1085.909,-29.210,444.520,174.427,18.301,152.983
C00669=1085.915,-28.960,444.508,174.429,18.302,152.983
C00670=1085.921,-28.711,444.494,174.430,18.304,152.983
C00671=1085.927,-28.461,444.482,174.432,18.305,152.983
C00672=1085.933,-28.211,444.469,174.433,18.307,152.983
C00673=1085.939,-27.961,444.457,174.435,18.309,152.983
C00674=1085.945,-27.712,444.444,174.437,18.311,152.983
C00675=1085.950,-27.463,444.431,174.438,18.312,152.983
C00676=1085.956,-27.213,444.419,174.440,18.314,152.983
C00677=1085.962,-26.963,444.406,174.441,18.316,152.983
C00678=1085.968,-26.714,444.393,174.442,18.317,152.984
C00679=1085.974,-26.464,444.380,174.444,18.319,152.984
C00680=1085.980,-26.214,444.368,174.446,18.321,152.984
C00681=1085.986,-25.965,444.355,174.447,18.323,152.984
C00682=1085.991,-25.715,444.342,174.448,18.325,152.984
C00683=1085.997,-25.466,444.329,174.450,18.326,152.984
C00684=1086.003,-25.216,444.316,174.452,18.328,152.984
C00685=1086.009,-24.966,444.303,174.453,18.330,152.984
C00686=1086.015,-24.717,444.291,174.455,18.331,152.984
C00687=1086.021,-24.467,444.278,174.456,18.333,152.984
C00688=1086.026,-24.218,444.265,174.457,18.335,152.984
C00689=1086.031,-23.968,444.252,174.459,18.337,152.984
C00690=1086.038,-23.719,444.239,174.461,18.339,152.984
C00691=1086.043,-23.469,444.226,174.463,18.340,152.984
C00692=1086.049,-23.219,444.214,174.464,18.342,152.984
C00693=1086.056,-22.970,444.201,174.465,18.344,152.984
C00694=1086.062,-22.720,444.188,174.467,18.345,152.984
C00695=1086.068,-22.470,444.175,174.469,18.347,152.984
C00696=1086.072,-22.221,444.162,174.470,18.349,152.985
C00697=1086.079,-21.972,444.149,174.471,18.351,152.985
C00698=1086.084,-21.722,444.136,174.473,18.353,152.985
C00699=1086.090,-21.472,444.124,174.474,18.354,152.985
C00700=1086.097,-21.223,444.110,174.476,18.356,152.985
C00701=1086.102,-20.972,444.097,174.478,18.358,152.985
C00702=1086.108,-20.723,444.084,174.479,18.360,152.985
C00703=1086.114,-20.473,444.071,174.480,18.361,152.985
C00704=1086.120,-20.224,444.058,174.482,18.363,152.985
C00705=1086.126,-19.974,444.046,174.484,18.365,152.985
C00706=1086.131,-19.725,444.032,174.485,18.367,152.985
C00707=1086.137,-19.475,444.019,174.487,18.369,152.985
C00708=1086.144,-19.225,444.006,174.488,18.370,152.985
C00709=1086.149,-18.976,443.994,174.489,18.372,152.985
C00710=1086.155,-18.727,443.980,174.492,18.374,152.985
C00711=1086.160,-18.477,443.967,174.493,18.375,152.985
C00712=1086.166,-18.228,443.954,174.494,18.377,152.986
C00713=1086.172,-17.978,443.941,174.496,18.379,152.986
C00714=1086.179,-17.728,443.928,174.497,18.381,152.986
C00715=1086.185,-17.479,443.915,174.499,18.383,152.986
C00716=1086.191,-17.206,443.901,174.501,18.384,152.986
C00717=1086.198,-16.933,443.886,174.502,18.386,152.986
C00718=1086.204,-16.660,443.872,174.504,18.388,152.986
C00719=1086.210,-16.388,443.858,174.506,18.390,152.986
C00720=1086.216,-16.138,443.844,174.508,18.392,152.986
C00721=1086.222,-15.889,443.832,174.509,18.394,152.986
C00722=1086.228,-15.639,443.818,174.510,18.396,152.986
C00723=1086.234,-15.390,443.805,174.512,18.397,152.986
C00724=1086.240,-15.140,443.792,174.513,18.399,152.986
C00725=1086.246,-14.891,443.779,174.515,18.401,152.986
C00726=1086.251,-14.640,443.766,174.517,18.403,152.986
C00727=1086.257,-14.391,443.752,174.518,18.404,152.986
C00728=1086.263,-14.142,443.739,174.520,18.406,152.987
C00729=1086.269,-13.892,443.726,174.521,18.408,152.987
C00730=1086.274,-13.642,443.712,174.523,18.410,152.987
C00731=1086.280,-13.393,443.699,174.524,18.412,152.987
C00732=1086.286,-13.143,443.686,174.526,18.413,152.987
C00733=1086.292,-12.893,443.672,174.527,18.415,152.987
C00734=1086.298,-12.644,443.659,174.529,18.417,152.987
C00735=1086.304,-12.395,443.645,174.531,18.419,152.987
C00736=1086.309,-12.145,443.633,174.532,18.420,152.987
C00737=1086.315,-11.895,443.619,174.533,18.422,152.987
C00738=1086.321,-11.646,443.606,174.535,18.425,152.987
C00739=1086.327,-11.396,443.593,174.537,18.426,152.987
C00740=1086.333,-11.146,443.579,174.538,18.428,152.987
C00741=1086.339,-10.897,443.566,174.539,18.430,152.988
C00742=1086.344,-10.648,443.552,174.541,18.431,152.988
C00743=1086.350,-10.398,443.539,174.543,18.433,152.988
C00744=1086.356,-10.148,443.526,174.544,18.435,152.988
C00745=1086.362,-9.899,443.512,174.546,18.437,152.988
C00746=1086.367,-9.649,443.498,174.547,18.438,152.988
C00747=1086.374,-9.400,443.485,174.549,18.441,152.988
C00748=1086.379,-9.150,443.472,174.550,18.443,152.988
C00749=1086.385,-8.901,443.459,174.552,18.444,152.988
C00750=1086.390,-8.651,443.445,174.553,18.446,152.988
C00751=1086.397,-8.402,443.432,174.556,18.448,152.988
C00752=1086.402,-8.152,443.418,174.557,18.450,152.988
C00753=1086.409,-7.902,443.404,174.558,18.451,152.988
C00754=1086.414,-7.652,443.391,174.560,18.453,152.988
C00755=1086.420,-7.403,443.378,174.562,18.455,152.988
C00756=1086.426,-7.153,443.364,174.563,18.457,152.989
C00757=1086.432,-6.904,443.351,174.564,18.459,152.989
C00758=1086.437,-6.654,443.337,174.566,18.460,152.989
C00759=1086.444,-6.405,443.323,174.567,18.462,152.989
C00760=1086.449,-6.155,443.310,174.569,18.464,152.989
C00761=1086.455,-5.906,443.296,174.571,18.466,152.989
C00762=1086.461,-5.655,443.283,174.572,18.467,152.989
C00763=1086.467,-5.406,443.270,174.573,18.469,152.989
C00764=1086.473,-5.156,443.256,174.576,18.471,152.989
C00765=1086.479,-4.907,443.242,174.577,18.473,152.989
C00766=1086.485,-4.658,443.229,174.578,18.475,152.989
C00767=1086.491,-4.408,443.215,174.580,18.476,152.989
C00768=1086.496,-4.159,443.201,174.582,18.478,152.989
C00769=1086.502,-3.909,443.188,174.583,18.480,152.989
C00770=1086.508,-3.659,443.174,174.585,18.482,152.989
C00771=1086.515,-3.410,443.161,174.586,18.483,152.990
C00772=1086.520,-3.160,443.147,174.588,18.485,152.989
C00773=1086.526,-2.911,443.133,174.589,18.488,152.990
C00774=1086.531,-2.661,443.119,174.591,18.489,152.990
C00775=1086.537,-2.412,443.106,174.593,18.491,152.990
C00776=1086.543,-2.162,443.092,174.594,18.493,152.990
C00777=1086.548,-1.913,443.078,174.596,18.495,152.990
C00778=1086.554,-1.663,443.064,174.597,18.496,152.990
C00779=1086.561,-1.413,443.051,174.599,18.499,152.990
C00780=1086.567,-1.140,443.035,174.601,18.500,152.990
C00781=1086.573,-0.865,443.020,174.603,18.503,152.990
C00782=1086.579,-0.591,443.005,174.604,18.505,152.990
C00783=1086.586,-0.316,442.990,174.606,18.507,152.991
C00784=1086.591,-0.067,442.976,174.607,18.509,152.991
C00785=1086.597,0.183,442.962,174.609,18.510,152.991
C00786=1086.602,0.432,442.948,174.610,18.512,152.991
C00787=1086.608,0.682,442.935,174.612,18.514,152.991
C00788=1086.614,0.932,442.921,174.614,18.516,152.991
C00789=1086.620,1.181,442.907,174.615,18.517,152.991
C00790=1086.625,1.431,442.893,174.616,18.520,152.991
C00791=1086.631,1.680,442.878,174.618,18.522,152.991
C00792=1086.637,1.929,442.865,174.620,18.523,152.991
C00793=1086.643,2.179,442.851,174.621,18.525,152.991
C00794=1086.649,2.429,442.837,174.622,18.527,152.991
C00795=1086.654,2.679,442.823,174.625,18.529,152.991
C00796=1086.660,2.928,442.809,174.626,18.531,152.992
C00797=1086.666,3.177,442.796,174.627,18.532,152.992
C00798=1086.672,3.426,442.781,174.630,18.535,152.992
C00799=1086.677,3.676,442.768,174.631,18.536,152.992
C00800=1086.683,3.926,442.753,174.632,18.538,152.992
C00801=1086.689,4.176,442.739,174.634,18.540,152.992
C00802=1086.694,4.425,442.726,174.636,18.542,152.992
C00803=1086.701,4.674,442.712,174.637,18.544,152.992
C00804=1086.707,4.924,442.697,174.638,18.545,152.992
C00805=1086.712,5.174,442.683,174.641,18.547,152.992
C00806=1086.718,5.424,442.670,174.642,18.549,152.992
C00807=1086.724,5.672,442.655,174.643,18.551,152.992
C00808=1086.729,5.922,442.641,174.645,18.553,152.992
C00809=1086.735,6.172,442.627,174.647,18.555,152.992
C00810=1086.741,6.422,442.614,174.648,18.557,152.993
C00811=1086.747,6.671,442.599,174.650,18.558,152.993
C00812=1086.753,6.920,442.585,174.652,18.560,152.993
C00813=1086.759,7.170,442.571,174.653,18.562,152.993
C00814=1086.764,7.420,442.557,174.654,18.564,152.993
C00815=1086.770,7.669,442.543,174.656,18.565,152.993
C00816=1086.776,7.919,442.528,174.658,18.568,152.993
C00817=1086.782,8.169,442.514,174.659,18.569,152.993
C00818=1086.788,8.417,442.500,174.661,18.571,152.993
C00819=1086.794,8.667,442.487,174.663,18.573,152.993
C00820=1086.800,8.917,442.472,174.664,18.575,152.993
C00821=1086.805,9.166,442.458,174.665,18.577,152.993
C00822=1086.811,9.416,442.444,174.667,18.578,152.993
C00823=1086.817,9.665,442.429,174.669,18.580,152.993
C00824=1086.823,9.915,442.415,174.671,18.582,152.993
C00825=1086.828,10.165,442.401,174.672,18.584,152.994
C00826=1086.835,10.414,442.386,174.674,18.586,152.994
C00827=1086.840,10.664,442.372,174.675,18.588,152.994
C00828=1086.846,10.913,442.359,174.677,18.589,152.994
C00829=1086.853,11.163,442.344,174.679,18.591,152.994
C00830=1086.858,11.412,442.330,174.680,18.593,152.994
C00831=1086.864,11.661,442.316,174.682,18.595,152.994
C00832=1086.870,11.912,442.302,174.683,18.596,152.994
C00833=1086.876,12.161,442.287,174.685,18.598,152.994
C00834=1086.881,12.410,442.273,174.687,18.600,152.994
C00835=1086.888,12.660,442.258,174.688,18.602,152.994
C00836=1086.893,12.909,442.244,174.690,18.604,152.994
C00837=1086.899,13.158,442.230,174.692,18.606,152.994
C00838=1086.905,13.409,442.215,174.693,18.608,152.994
C00839=1086.911,13.658,442.201,174.695,18.610,152.994
C00840=1086.917,13.908,442.187,174.697,18.611,152.994
C00841=1086.923,14.157,442.172,174.698,18.613,152.995
C00842=1086.928,14.406,442.158,174.699,18.614,152.995
C00843=1086.934,14.656,442.143,174.701,18.617,152.995
C00844=1086.941,14.932,442.127,174.703,18.619,152.995
C00845=1086.947,15.208,442.112,174.705,18.621,152.995
C00846=1086.954,15.485,442.095,174.706,18.623,152.995
C00847=1086.960,15.761,442.080,174.708,18.625,152.995
C00848=1086.965,16.011,442.066,174.710,18.627,152.995
C00849=1086.972,16.260,442.051,174.712,18.629,152.995
C00850=1086.977,16.510,442.037,174.713,18.630,152.995
C00851=1086.982,16.759,442.022,174.715,18.632,152.995
C00852=1086.989,17.009,442.007,174.717,18.634,152.995
C00853=1086.994,17.258,441.993,174.718,18.636,152.995
C00854=1087.000,17.508,441.978,174.720,18.638,152.995
C00855=1087.006,17.757,441.964,174.722,18.640,152.996
C00856=1087.012,18.006,441.950,174.723,18.642,152.996
C00857=1087.018,18.256,441.935,174.724,18.643,152.996
C00858=1087.023,18.506,441.920,174.726,18.645,152.996
C00859=1087.029,18.756,441.905,174.728,18.647,152.996
C00860=1087.035,19.005,441.891,174.729,18.649,152.996
C00861=1087.040,19.254,441.877,174.731,18.650,152.996
C00862=1087.047,19.504,441.862,174.733,18.652,152.996
C00863=1087.053,19.753,441.847,174.734,18.655,152.996
C00864=1087.058,20.003,441.832,174.736,18.656,152.996
C00865=1087.064,20.252,441.818,174.738,18.658,152.996
C00866=1087.070,20.501,441.803,174.739,18.660,152.996
C00867=1087.076,20.752,441.789,174.740,18.662,152.996
C00868=1087.081,21.001,441.774,174.743,18.664,152.996
C00869=1087.087,21.250,441.759,174.744,18.665,152.996
C00870=1087.093,21.499,441.744,174.746,18.667,152.997
C00871=1087.098,21.750,441.730,174.748,18.669,152.997
C00872=1087.104,21.999,441.715,174.749,18.671,152.997
C00873=1087.110,22.248,441.700,174.750,18.673,152.997
C00874=1087.116,22.498,441.685,174.753,18.675,152.997
C00875=1087.121,22.747,441.671,174.754,18.677,152.997
C00876=1087.127,22.997,441.656,174.755,18.678,152.997
C00877=1087.133,23.246,441.641,174.758,18.680,152.997
C00878=1087.139,23.496,441.626,174.759,18.682,152.997
C00879=1087.144,23.745,441.611,174.760,18.684,152.997
C00880=1087.151,23.995,441.597,174.762,18.686,152.997
C00881=1087.156,24.245,441.582,174.764,18.687,152.997
C00882=1087.162,24.494,441.567,174.765,18.689,152.997
C00883=1087.168,24.743,441.552,174.767,18.692,152.997
C00884=1087.174,24.992,441.538,174.769,18.693,152.998
C00885=1087.179,25.242,441.522,174.770,18.695,152.998
C00886=1087.185,25.492,441.508,174.772,18.697,152.998
C00887=1087.191,25.741,441.493,174.774,18.698,152.998
C00888=1087.196,25.991,441.478,174.776,18.701,152.998
C00889=1087.202,26.240,441.463,174.777,18.702,152.998
C00890=1087.208,26.490,441.448,174.779,18.704,152.998
C00891=1087.214,26.739,441.433,174.781,18.706,152.998
C00892=1087.220,26.988,441.419,174.782,18.707,152.998
C00893=1087.225,27.238,441.403,174.784,18.710,152.998
C00894=1087.232,27.488,441.388,174.786,18.712,152.998
C00895=1087.237,27.737,441.374,174.787,18.713,152.998
C00896=1087.243,27.987,441.359,174.789,18.715,152.998
C00897=1087.249,28.236,441.344,174.791,18.717,152.998
C00898=1087.254,28.486,441.329,174.792,18.719,152.998
C00899=1087.260,28.735,441.314,174.794,18.720,152.998
C00900=1087.266,28.985,441.299,174.796,18.722,152.998
C00901=1087.271,29.234,441.284,174.797,18.724,152.998
C00902=1087.277,29.484,441.268,174.798,18.726,152.999
C00903=1087.283,29.733,441.254,174.801,18.728,152.999
C00904=1087.289,29.983,441.238,174.802,18.730,152.999
C00905=1087.294,30.232,441.224,174.804,18.732,152.999
C00906=1087.300,30.482,441.208,174.806,18.734,152.999
C00907=1087.306,30.731,441.194,174.807,18.735,152.999
C00908=1087.312,31.009,441.176,174.809,18.737,152.999
C00909=1087.319,31.286,441.159,174.811,18.740,152.999
C00910=1087.325,31.564,441.142,174.813,18.741,152.999
C00911=1087.331,31.842,441.126,174.815,18.743,152.999
C00912=1087.336,32.091,441.111,174.816,18.745,152.999
C00913=1087.343,32.341,441.096,174.818,18.748,152.999
C00914=1087.349,32.590,441.080,174.820,18.749,152.999
C00915=1087.355,32.839,441.065,174.821,18.751,152.999
C00916=1087.360,33.089,441.050,174.824,18.753,152.999
C00917=1087.366,33.338,441.035,174.825,18.754,152.999
C00918=1087.372,33.588,441.019,174.826,18.756,153.000
C00919=1087.377,33.837,441.005,174.828,18.758,153.000
C00920=1087.383,34.087,440.989,174.830,18.760,153.000
C00921=1087.389,34.337,440.974,174.831,18.761,153.000
C00922=1087.395,34.586,440.959,174.834,18.763,153.000
C00923=1087.400,34.835,440.943,174.835,18.766,153.000
C00924=1087.406,35.084,440.928,174.837,18.768,153.000
C00925=1087.412,35.334,440.913,174.838,18.769,153.000
C00926=1087.418,35.584,440.898,174.840,18.771,153.000
C00927=1087.423,35.833,440.883,174.842,18.773,153.000
C00928=1087.429,36.082,440.866,174.843,18.774,153.000
C00929=1087.436,36.332,440.851,174.845,18.776,153.000
C00930=1087.441,36.581,440.836,174.847,18.778,153.000
C00931=1087.447,36.831,440.821,174.848,18.780,153.000
C00932=1087.453,37.081,440.806,174.851,18.782,153.000
C00933=1087.458,37.330,440.790,174.852,18.783,153.000
C00934=1087.464,37.579,440.775,174.853,18.785,153.000
C00935=1087.470,37.829,440.759,174.856,18.787,153.000
C00936=1087.475,38.079,440.744,174.857,18.789,153.001
C00937=1087.482,38.328,440.729,174.859,18.791,153.001
C00938=1087.487,38.577,440.713,174.861,18.793,153.001
C00939=1087.493,38.827,440.698,174.862,18.794,153.001
C00940=1087.498,39.077,440.682,174.864,18.796,153.001
C00941=1087.504,39.325,440.667,174.866,18.798,153.001
C00942=1087.510,39.575,440.651,174.868,18.800,153.001
C00943=1087.516,39.825,440.636,174.869,18.802,153.001
C00944=1087.521,40.074,440.620,174.871,18.804,153.001
C00945=1087.527,40.324,440.605,174.873,18.806,153.001
C00946=1087.533,40.573,440.590,174.874,18.807,153.001
C00947=1087.538,40.822,440.574,174.877,18.809,153.001
C00948=1087.544,41.072,440.558,174.878,18.811,153.001
C00949=1087.550,41.322,440.543,174.879,18.813,153.001
C00950=1087.556,41.570,440.527,174.881,18.815,153.001
C00951=1087.561,41.820,440.512,174.883,18.816,153.001
C00952=1087.567,42.070,440.496,174.884,18.818,153.001
C00953=1087.572,42.319,440.480,174.887,18.820,153.001
C00954=1087.578,42.569,440.465,174.888,18.821,153.001
C00955=1087.585,42.818,440.449,174.890,18.824,153.002
C00956=1087.590,43.067,440.434,174.891,18.826,153.002
C00957=1087.596,43.316,440.418,174.894,18.828,153.002
C00958=1087.601,43.566,440.402,174.895,18.829,153.002
C00959=1087.607,43.816,440.387,174.897,18.831,153.002
C00960=1087.612,44.065,440.371,174.899,18.833,153.002
C00961=1087.618,44.315,440.355,174.900,18.834,153.002
C00962=1087.624,44.564,440.339,174.902,18.837,153.002
C00963=1087.629,44.814,440.324,174.904,18.838,153.002
C00964=1087.635,45.063,440.307,174.905,18.840,153.002
C00965=1087.641,45.313,440.292,174.907,18.842,153.002
C00966=1087.646,45.562,440.276,174.909,18.843,153.002
C00967=1087.652,45.812,440.261,174.911,18.846,153.002
C00968=1087.657,46.061,440.244,174.912,18.848,153.002
C00969=1087.662,46.310,440.229,174.914,18.849,153.002
C00970=1087.668,46.560,440.213,174.916,18.851,153.002
C00971=1087.674,46.810,440.197,174.917,18.853,153.002
C00972=1087.681,47.087,440.179,174.920,18.855,153.002
C00973=1087.686,47.364,440.162,174.922,18.857,153.003
C00974=1087.693,47.642,440.145,174.923,18.859,153.003
C00975=1087.699,47.920,440.127,174.925,18.861,153.003
C00976=1087.705,48.169,440.111,174.927,18.862,153.003
C00977=1087.711,48.419,440.095,174.929,18.865,153.003
C00978=1087.716,48.669,440.079,174.931,18.866,153.003
C00979=1087.722,48.917,440.063,174.933,18.869,153.003
C00980=1087.727,49.167,440.048,174.934,18.870,153.003
C00981=1087.733,49.417,440.031,174.936,18.872,153.003
C00982=1087.739,49.666,440.015,174.938,18.874,153.003
C00983=1087.744,49.915,440.000,174.939,18.875,153.003
C00984=1087.750,50.165,439.984,174.941,18.877,153.003
C00985=1087.756,50.414,439.967,174.943,18.879,153.003
C00986=1087.762,50.664,439.952,174.945,18.881,153.003
C00987=1087.767,50.913,439.936,174.947,18.882,153.003
C00988=1087.773,51.162,439.920,174.949,18.884,153.003
C00989=1087.779,51.412,439.904,174.950,18.886,153.003
C00990=1087.784,51.662,439.887,174.952,18.888,153.003
C00991=1087.790,51.911,439.871,174.954,18.890,153.003
C00992=1087.795,52.160,439.856,174.955,18.892,153.003
C00993=1087.801,52.410,439.840,174.957,18.894,153.003
C00994=1087.807,52.659,439.823,174.959,18.895,153.003
C00995=1087.813,52.908,439.807,174.961,18.897,153.003
C00996=1087.819,53.158,439.792,174.963,18.899,153.004
C00997=1087.825,53.408,439.775,174.965,18.901,153.004
C00998=1087.830,53.656,439.759,174.966,18.902,153.004
C00999=1087.836,53.906,439.743,174.968,18.904,153.004
C01000=1087.842,54.156,439.728,174.970,18.906,153.004
C01001=1087.847,54.405,439.711,174.971,18.908,153.004
C01002=1087.853,54.655,439.695,174.974,18.910,153.004
C01003=1087.859,54.904,439.678,174.975,18.911,153.004
C01004=1087.865,55.153,439.662,174.977,18.913,153.004
C01005=1087.870,55.402,439.647,174.979,18.915,153.004
C01006=1087.876,55.652,439.631,174.980,18.916,153.004
C01007=1087.882,55.901,439.614,174.983,18.918,153.004
C01008=1087.887,56.151,439.598,174.984,18.920,153.004
C01009=1087.893,56.400,439.581,174.986,18.922,153.004
C01010=1087.899,56.650,439.565,174.988,18.923,153.004
C01011=1087.905,56.899,439.549,174.990,18.925,153.004
C01012=1087.910,57.149,439.533,174.991,18.927,153.004
C01013=1087.916,57.398,439.517,174.994,18.929,153.004
C01014=1087.922,57.648,439.501,174.995,18.931,153.004
C01015=1087.927,57.897,439.484,174.997,18.933,153.004
C01016=1087.933,58.146,439.468,174.999,18.934,153.004
C01017=1087.939,58.395,439.452,175.001,18.935,153.004
C01018=1087.945,58.645,439.435,175.003,18.937,153.004
C01019=1087.951,58.894,439.419,175.004,18.939,153.004
C01020=1087.956,59.143,439.403,175.007,18.941,153.004
C01021=1087.962,59.393,439.386,175.008,18.942,153.004
C01022=1087.968,59.642,439.370,175.010,18.944,153.004
C01023=1087.974,59.892,439.354,175.012,18.946,153.004
C01024=1087.980,60.141,439.337,175.014,18.948,153.004
C01025=1087.986,60.390,439.321,175.015,18.949,153.004
C01026=1087.991,60.640,439.304,175.018,18.952,153.004
C01027=1087.997,60.889,439.288,175.019,18.953,153.004
C01028=1088.003,61.139,439.272,175.021,18.954,153.004
C01029=1088.009,61.388,439.255,175.023,18.956,153.004
C01030=1088.015,61.637,439.239,175.024,18.958,153.004
C01031=1088.020,61.887,439.222,175.027,18.960,153.004
C01032=1088.026,62.136,439.206,175.028,18.961,153.004
C01033=1088.032,62.386,439.190,175.030,18.963,153.004
C01034=1088.038,62.635,439.174,175.032,18.965,153.004
C01035=1088.044,62.884,439.157,175.034,18.966,153.004
C01036=1088.050,63.162,439.139,175.036,18.968,153.004
C01037=1088.056,63.439,439.120,175.038,18.970,153.004
C01038=1088.062,63.717,439.102,175.040,18.972,153.004
C01039=1088.069,63.994,439.084,175.043,18.974,153.004
C01040=1088.075,64.244,439.067,175.044,18.976,153.004
C01041=1088.081,64.494,439.051,175.046,18.978,153.004
C01042=1088.087,64.743,439.034,175.048,18.979,153.004
C01043=1088.092,64.992,439.017,175.050,18.981,153.004
C01044=1088.098,65.242,439.001,175.052,18.982,153.004
C01045=1088.104,65.491,438.984,175.053,18.984,153.004
C01046=1088.110,65.741,438.967,175.055,18.986,153.004
C01047=1088.115,65.990,438.951,175.057,18.987,153.004
C01048=1088.121,66.240,438.934,175.059,18.989,153.004
C01049=1088.127,66.488,438.917,175.061,18.991,153.004
C01050=1088.132,66.738,438.900,175.063,18.993,153.004
C01051=1088.138,66.987,438.884,175.064,18.995,153.005
C01052=1088.143,67.237,438.867,175.067,18.996,153.004
C01053=1088.149,67.486,438.851,175.068,18.998,153.004
C01054=1088.155,67.735,438.834,175.071,19.000,153.004
C01055=1088.161,67.985,438.817,175.072,19.001,153.005
C01056=1088.166,68.234,438.800,175.074,19.003,153.005
C01057=1088.172,68.484,438.784,175.076,19.005,153.005
C01058=1088.177,68.733,438.767,175.078,19.007,153.005
C01059=1088.183,68.982,438.750,175.080,19.008,153.004
C01060=1088.189,69.232,438.734,175.082,19.010,153.004
C01061=1088.195,69.480,438.717,175.083,19.011,153.005
C01062=1088.200,69.730,438.700,175.086,19.013,153.005
C01063=1088.206,69.979,438.683,175.087,19.015,153.005
C01064=1088.211,70.229,438.667,175.089,19.017,153.005
C01065=1088.217,70.478,438.650,175.091,19.018,153.005
C01066=1088.223,70.727,438.633,175.093,19.020,153.005
C01067=1088.229,70.978,438.616,175.095,19.022,153.005
C01068=1088.235,71.227,438.599,175.097,19.024,153.005
C01069=1088.240,71.476,438.582,175.099,19.025,153.005
C01070=1088.246,71.725,438.565,175.101,19.027,153.005
C01071=1088.251,71.975,438.548,175.102,19.028,153.005
C01072=1088.257,72.224,438.532,175.105,19.030,153.005
C01073=1088.263,72.473,438.514,175.106,19.032,153.005
C01074=1088.268,72.723,438.497,175.108,19.034,153.005
C01075=1088.274,72.971,438.480,175.110,19.035,153.005
C01076=1088.280,73.221,438.463,175.112,19.037,153.005
C01077=1088.285,73.471,438.447,175.114,19.038,153.005
C01078=1088.291,73.719,438.430,175.116,19.041,153.005
C01079=1088.297,73.970,438.412,175.118,19.042,153.005
C01080=1088.302,74.219,438.395,175.120,19.044,153.004
C01081=1088.308,74.468,438.379,175.122,19.045,153.005
C01082=1088.314,74.717,438.361,175.124,19.047,153.005
C01083=1088.319,74.967,438.344,175.125,19.049,153.005
C01084=1088.325,75.216,438.327,175.128,19.051,153.005
C01085=1088.331,75.465,438.310,175.129,19.052,153.005
C01086=1088.337,75.715,438.292,175.132,19.054,153.005
C01087=1088.343,75.964,438.276,175.133,19.055,153.005
C01088=1088.348,76.213,438.259,175.135,19.057,153.004
C01089=1088.353,76.463,438.242,175.137,19.058,153.005
C01090=1088.360,76.712,438.225,175.139,19.060,153.005
C01091=1088.365,76.961,438.208,175.141,19.062,153.005
C01092=1088.371,77.211,438.190,175.143,19.064,153.004
C01093=1088.377,77.461,438.174,175.145,19.065,153.004
C01094=1088.382,77.710,438.156,175.147,19.067,153.004
C01095=1088.388,77.959,438.139,175.149,19.068,153.004
C01096=1088.393,78.208,438.122,175.151,19.070,153.004
C01097=1088.399,78.457,438.105,175.152,19.072,153.004
C01098=1088.405,78.707,438.087,175.155,19.074,153.004
C01099=1088.411,78.956,438.070,175.156,19.075,153.004
C01100=1088.417,79.233,438.051,175.159,19.077,153.004
C01101=1088.423,79.511,438.032,175.161,19.079,153.004
C01102=1088.430,79.789,438.012,175.163,19.081,153.004
C01103=1088.435,80.066,437.993,175.165,19.083,153.004
C01104=1088.441,80.316,437.976,175.167,19.084,153.004
C01105=1088.447,80.564,437.959,175.169,19.086,153.004
C01106=1088.452,80.814,437.942,175.171,19.088,153.004
C01107=1088.458,81.064,437.924,175.173,19.089,153.004
C01108=1088.464,81.313,437.906,175.175,19.091,153.004
C01109=1088.469,81.562,437.889,175.177,19.093,153.004
C01110=1088.475,81.811,437.872,175.178,19.094,153.004
C01111=1088.480,82.060,437.854,175.181,19.096,153.004
C01112=1088.486,82.310,437.836,175.183,19.098,153.004
C01113=1088.492,82.560,437.819,175.185,19.099,153.004
C01114=1088.497,82.809,437.802,175.187,19.101,153.004
C01115=1088.503,83.058,437.784,175.189,19.102,153.004
C01116=1088.508,83.307,437.767,175.191,19.104,153.004
C01117=1088.515,83.557,437.750,175.193,19.105,153.004
C01118=1088.520,83.806,437.733,175.195,19.107,153.004
C01119=1088.526,84.055,437.715,175.196,19.109,153.004
C01120=1088.531,84.304,437.697,175.199,19.111,153.004
C01121=1088.537,84.554,437.679,175.200,19.112,153.004
C01122=1088.543,84.804,437.663,175.203,19.114,153.004
C01123=1088.548,85.053,437.645,175.204,19.115,153.004
C01124=1088.554,85.302,437.627,175.207,19.117,153.004
C01125=1088.560,85.551,437.610,175.209,19.119,153.004
C01126=1088.565,85.800,437.592,175.211,19.120,153.004
C01127=1088.571,86.049,437.574,175.213,19.122,153.004
C01128=1088.577,86.299,437.556,175.214,19.123,153.004
C01129=1088.582,86.549,437.540,175.217,19.125,153.004
C01130=1088.588,86.798,437.522,175.218,19.126,153.004
C01131=1088.594,87.048,437.504,175.221,19.128,153.004
C01132=1088.599,87.297,437.487,175.222,19.129,153.004
C01133=1088.605,87.546,437.469,175.225,19.131,153.004
C01134=1088.611,87.795,437.451,175.227,19.133,153.004
C01135=1088.616,88.044,437.434,175.229,19.135,153.004
C01136=1088.622,88.294,437.416,175.231,19.137,153.004
C01137=1088.628,88.543,437.398,175.233,19.138,153.004
C01138=1088.634,88.792,437.380,175.235,19.140,153.004
C01139=1088.639,89.041,437.363,175.237,19.141,153.003
C01140=1088.645,89.291,437.345,175.239,19.143,153.003
C01141=1088.651,89.540,437.327,175.241,19.144,153.003
C01142=1088.656,89.789,437.310,175.243,19.146,153.003
C01143=1088.662,90.039,437.292,175.245,19.147,153.003
C01144=1088.668,90.288,437.274,175.247,19.149,153.003
C01145=1088.674,90.538,437.256,175.249,19.150,153.003
C01146=1088.679,90.787,437.239,175.251,19.152,153.003
C01147=1088.685,91.036,437.221,175.253,19.153,153.003
C01148=1088.691,91.286,437.203,175.255,19.155,153.003
C01149=1088.696,91.535,437.185,175.257,19.157,153.003
C01150=1088.701,91.784,437.168,175.260,19.159,153.003
C01151=1088.708,92.034,437.150,175.261,19.160,153.003
C01152=1088.713,92.283,437.132,175.264,19.162,153.003
C01153=1088.719,92.532,437.115,175.265,19.163,153.003
C01154=1088.724,92.782,437.096,175.268,19.165,153.003
C01155=1088.730,93.030,437.078,175.269,19.166,153.003
C01156=1088.735,93.279,437.060,175.271,19.168,153.003
C01157=1088.741,93.529,437.042,175.274,19.169,153.003
C01158=1088.746,93.778,437.024,175.275,19.171,153.003
C01159=1088.752,94.028,437.006,175.278,19.172,153.003
C01160=1088.758,94.277,436.989,175.279,19.174,153.003
C01161=1088.763,94.526,436.971,175.282,19.175,153.002
C01162=1088.770,94.775,436.952,175.283,19.177,153.003
C01163=1088.775,95.025,436.934,175.286,19.178,153.002
C01164=1088.781,95.303,436.914,175.288,19.181,153.002
C01165=1088.787,95.580,436.894,175.291,19.182,153.002
C01166=1088.794,95.857,436.875,175.293,19.184,153.002
C01167=1088.800,96.135,436.855,175.296,19.186,153.002
C01168=1088.805,96.384,436.836,175.297,19.187,153.002
C01169=1088.811,96.633,436.818,175.300,19.189,153.002
C01170=1088.817,96.883,436.800,175.301,19.190,153.002
C01171=1088.823,97.132,436.783,175.303,19.192,153.002
C01172=1088.828,97.381,436.763,175.305,19.193,153.002
C01173=1088.834,97.630,436.746,175.307,19.195,153.002
C01174=1088.840,97.880,436.728,175.310,19.196,153.002
C01175=1088.845,98.129,436.709,175.311,19.198,153.002
C01176=1088.851,98.378,436.691,175.314,19.199,153.002
C01177=1088.857,98.627,436.674,175.316,19.200,153.002
C01178=1088.862,98.877,436.655,175.318,19.202,153.002
C01179=1088.868,99.126,436.637,175.320,19.204,153.002
C01180=1088.874,99.376,436.619,175.322,19.206,153.002
C01181=1088.879,99.625,436.601,175.324,19.207,153.001
C01182=1088.885,99.874,436.582,175.326,19.208,153.001
C01183=1088.891,100.123,436.564,175.328,19.210,153.001
C01184=1088.897,100.372,436.546,175.331,19.212,153.001
C01185=1088.902,100.622,436.528,175.333,19.213,153.001
C01186=1088.908,100.871,436.510,175.335,19.215,153.001
C01187=1088.914,101.120,436.491,175.337,19.216,153.001
C01188=1088.919,101.370,436.473,175.339,19.217,153.001
C01189=1088.925,101.618,436.455,175.341,19.219,153.001
C01190=1088.930,101.868,436.436,175.343,19.220,153.001
C01191=1088.936,102.117,436.418,175.346,19.222,153.001
C01192=1088.942,102.367,436.399,175.347,19.223,153.001
C01193=1088.947,102.616,436.382,175.350,19.225,153.001
C01194=1088.953,102.865,436.362,175.352,19.226,153.001
C01195=1088.958,103.114,436.345,175.354,19.228,153.001
C01196=1088.964,103.364,436.326,175.356,19.230,153.000
C01197=1088.969,103.613,436.308,175.358,19.232,153.000
C01198=1088.975,103.862,436.289,175.360,19.233,153.000
C01199=1088.981,104.111,436.271,175.363,19.234,153.000
C01200=1088.986,104.361,436.252,175.364,19.236,153.000
C01201=1088.991,104.610,436.234,175.367,19.237,153.000
C01202=1088.998,104.859,436.215,175.369,19.239,153.000
C01203=1089.002,105.108,436.197,175.371,19.240,153.000
C01204=1089.009,105.358,436.178,175.373,19.242,153.000
C01205=1089.014,105.607,436.160,175.375,19.243,153.000
C01206=1089.020,105.856,436.142,175.377,19.244,153.000
C01207=1089.026,106.106,436.122,175.380,19.246,153.000
C01208=1089.031,106.355,436.105,175.381,19.247,153.000
C01209=1089.037,106.604,436.085,175.384,19.249,153.000
C01210=1089.042,106.853,436.067,175.386,19.251,152.999
C01211=1089.048,107.102,436.049,175.388,19.252,152.999
C01212=1089.053,107.351,436.030,175.390,19.254,152.999
C01213=1089.059,107.601,436.012,175.393,19.255,152.999
C01214=1089.065,107.850,435.993,175.395,19.256,152.999
C01215=1089.071,108.099,435.974,175.397,19.258,152.999
C01216=1089.076,108.349,435.956,175.398,19.259,152.999
C01217=1089.081,108.598,435.937,175.401,19.261,152.999
C01218=1089.088,108.847,435.918,175.404,19.262,152.999
C01219=1089.093,109.097,435.900,175.405,19.263,152.999
C01220=1089.099,109.345,435.881,175.408,19.265,152.999
C01221=1089.105,109.595,435.862,175.410,19.267,152.999
C01222=1089.110,109.845,435.844,175.412,19.268,152.998
C01223=1089.116,110.093,435.825,175.414,19.269,152.998
C01224=1089.122,110.343,435.806,175.416,19.270,152.998
C01225=1089.127,110.592,435.787,175.418,19.272,152.998
C01226=1089.133,110.841,435.769,175.421,19.274,152.998
C01227=1089.138,111.090,435.750,175.422,19.275,152.998
C01228=1089.145,111.368,435.729,175.425,19.277,152.998
C01229=1089.151,111.645,435.708,175.428,19.278,152.998
C01230=1089.158,111.923,435.687,175.430,19.280,152.998
C01231=1089.163,112.201,435.666,175.433,19.281,152.998
C01232=1089.169,112.449,435.648,175.435,19.283,152.998
C01233=1089.175,112.699,435.629,175.437,19.285,152.997
C01234=1089.181,112.948,435.609,175.439,19.286,152.997
C01235=1089.186,113.196,435.591,175.442,19.287,152.997
C01236=1089.192,113.446,435.573,175.443,19.288,152.997
C01237=1089.197,113.696,435.553,175.446,19.290,152.997
C01238=1089.203,113.945,435.534,175.448,19.291,152.997
C01239=1089.208,114.194,435.515,175.450,19.293,152.997
C01240=1089.215,114.443,435.497,175.452,19.294,152.997
C01241=1089.220,114.693,435.477,175.455,19.296,152.997
C01242=1089.225,114.941,435.459,175.457,19.297,152.997
C01243=1089.231,115.191,435.439,175.459,19.299,152.996
C01244=1089.237,115.440,435.420,175.462,19.300,152.996
C01245=1089.242,115.689,435.401,175.463,19.302,152.996
C01246=1089.247,115.939,435.383,175.466,19.303,152.996
C01247=1089.253,116.188,435.363,175.468,19.305,152.996
C01248=1089.258,116.437,435.345,175.470,19.306,152.996
C01249=1089.264,116.687,435.325,175.472,19.307,152.996
C01250=1089.269,116.936,435.306,175.475,19.309,152.996
C01251=1089.275,117.185,435.287,175.476,19.310,152.996
C01252=1089.280,117.434,435.268,175.479,19.312,152.996
C01253=1089.287,117.683,435.249,175.481,19.313,152.996
C01254=1089.292,117.932,435.230,175.483,19.314,152.995
C01255=1089.297,118.181,435.211,175.486,19.316,152.995
C01256=1089.303,118.431,435.192,175.488,19.318,152.995
C01257=1089.308,118.680,435.173,175.491,19.319,152.995
C01258=1089.314,118.929,435.154,175.492,19.320,152.995
C01259=1089.320,119.178,435.134,175.495,19.322,152.995
C01260=1089.326,119.427,435.115,175.497,19.324,152.995
C01261=1089.331,119.676,435.096,175.499,19.325,152.995
C01262=1089.336,119.925,435.076,175.501,19.326,152.995
C01263=1089.342,120.175,435.057,175.504,19.328,152.995
C01264=1089.348,120.424,435.038,175.506,19.329,152.994
C01265=1089.353,120.673,435.019,175.508,19.330,152.994
C01266=1089.359,120.923,435.000,175.511,19.332,152.994
C01267=1089.364,121.172,434.981,175.512,19.333,152.994
C01268=1089.370,121.421,434.961,175.515,19.334,152.994
C01269=1089.376,121.670,434.941,175.517,19.336,152.994
C01270=1089.381,121.919,434.923,175.519,19.337,152.994
C01271=1089.387,122.168,434.903,175.522,19.339,152.994
C01272=1089.392,122.418,434.884,175.524,19.340,152.994
C01273=1089.397,122.668,434.864,175.526,19.341,152.993
C01274=1089.403,122.916,434.844,175.528,19.343,152.993
C01275=1089.408,123.165,434.825,175.531,19.344,152.993
C01276=1089.414,123.415,434.806,175.533,19.346,152.993
C01277=1089.420,123.664,434.787,175.535,19.347,152.993
C01278=1089.426,123.913,434.767,175.538,19.348,152.993
C01279=1089.431,124.162,434.748,175.540,19.350,152.993
C01280=1089.437,124.412,434.728,175.542,19.351,152.993
C01281=1089.442,124.660,434.710,175.544,19.352,152.993
C01282=1089.448,124.909,434.690,175.547,19.353,152.992
C01283=1089.454,125.159,434.670,175.549,19.354,152.992
C01284=1089.460,125.408,434.651,175.551,19.356,152.992
C01285=1089.466,125.657,434.631,175.554,19.357,152.992
C01286=1089.471,125.906,434.612,175.556,19.359,152.992
C01287=1089.476,126.156,434.592,175.558,19.360,152.992
C01288=1089.482,126.405,434.572,175.561,19.362,152.992
C01289=1089.487,126.654,434.553,175.563,19.363,152.991
C01290=1089.493,126.903,434.534,175.565,19.364,152.991
C01291=1089.499,127.152,434.514,175.568,19.365,152.991
C01292=1089.506,127.430,434.492,175.570,19.367,152.991
C01293=1089.511,127.708,434.471,175.573,19.368,152.991
C01294=1089.518,127.985,434.449,175.575,19.370,152.991
C01295=1089.524,128.262,434.427,175.578,19.371,152.991
C01296=1089.530,128.511,434.407,175.580,19.373,152.990
C01297=1089.535,128.760,434.388,175.583,19.374,152.990
C01298=1089.541,129.009,434.368,175.585,19.375,152.990
C01299=1089.547,129.259,434.349,175.587,19.376,152.990
C01300=1089.553,129.508,434.329,175.590,19.378,152.990
C01301=1089.559,129.757,434.310,175.592,19.380,152.990
C01302=1089.564,130.007,434.290,175.594,19.380,152.990
C01303=1089.570,130.256,434.270,175.597,19.382,152.989
C01304=1089.575,130.505,434.251,175.599,19.383,152.989
C01305=1089.581,130.754,434.231,175.601,19.384,152.989
C01306=1089.587,131.003,434.211,175.604,19.385,152.989
C01307=1089.593,131.252,434.191,175.606,19.387,152.989
C01308=1089.598,131.501,434.171,175.609,19.388,152.989
C01309=1089.604,131.751,434.152,175.611,19.389,152.989
C01310=1089.610,131.999,434.132,175.613,19.390,152.988
C01311=1089.616,132.249,434.112,175.616,19.392,152.988
C01312=1089.621,132.498,434.092,175.618,19.393,152.988
C01313=1089.627,132.747,434.073,175.620,19.394,152.988
C01314=1089.633,132.996,434.053,175.623,19.396,152.988
C01315=1089.638,133.245,434.032,175.625,19.397,152.988
C01316=1089.644,133.495,434.013,175.628,19.399,152.987
C01317=1089.650,133.744,433.993,175.630,19.400,152.987
C01318=1089.654,133.993,433.973,175.632,19.401,152.987
C01319=1089.660,134.242,433.953,175.635,19.402,152.987
C01320=1089.666,134.491,433.932,175.637,19.403,152.987
C01321=1089.671,134.741,433.913,175.639,19.405,152.987
C01322=1089.677,134.989,433.893,175.642,19.406,152.987
C01323=1089.683,135.239,433.873,175.644,19.408,152.987
C01324=1089.688,135.488,433.853,175.646,19.408,152.986
C01325=1089.694,135.737,433.833,175.649,19.410,152.986
C01326=1089.700,135.986,433.813,175.651,19.411,152.986
C01327=1089.706,136.235,433.793,175.654,19.412,152.986
C01328=1089.711,136.485,433.773,175.657,19.414,152.986
C01329=1089.717,136.733,433.753,175.658,19.415,152.986
C01330=1089.722,136.982,433.733,175.661,19.417,152.985
C01331=1089.728,137.231,433.713,175.664,19.418,152.985
C01332=1089.733,137.481,433.693,175.666,19.419,152.985
C01333=1089.739,137.730,433.673,175.668,19.420,152.985
C01334=1089.744,137.979,433.652,175.671,19.421,152.985
C01335=1089.750,138.228,433.632,175.673,19.423,152.985
C01336=1089.756,138.477,433.612,175.676,19.424,152.984
C01337=1089.761,138.726,433.593,175.678,19.425,152.984
C01338=1089.767,138.975,433.573,175.680,19.426,152.984
C01339=1089.772,139.224,433.552,175.683,19.428,152.984
C01340=1089.777,139.473,433.532,175.685,19.429,152.984
C01341=1089.784,139.723,433.511,175.687,19.430,152.984
C01342=1089.789,139.972,433.491,175.690,19.431,152.984
C01343=1089.795,140.221,433.471,175.692,19.433,152.983
C01344=1089.800,140.471,433.451,175.695,19.434,152.983
C01345=1089.806,140.719,433.431,175.697,19.436,152.983
C01346=1089.811,140.969,433.410,175.699,19.436,152.983
C01347=1089.817,141.217,433.390,175.702,19.438,152.983
C01348=1089.823,141.466,433.370,175.704,19.439,152.983
C01349=1089.828,141.716,433.349,175.707,19.440,152.982
C01350=1089.834,141.964,433.329,175.709,19.441,152.982
C01351=1089.839,142.214,433.309,175.711,19.443,152.982
C01352=1089.845,142.463,433.288,175.714,19.444,152.982
C01353=1089.851,142.712,433.268,175.717,19.445,152.982
C01354=1089.856,142.961,433.247,175.720,19.446,152.981
C01355=1089.862,143.210,433.227,175.721,19.447,152.981
C01356=1089.868,143.487,433.205,175.724,19.449,152.981
C01357=1089.874,143.765,433.181,175.727,19.451,152.981
C01358=1089.880,144.042,433.159,175.730,19.452,152.981
C01359=1089.886,144.320,433.136,175.733,19.453,152.980
C01360=1089.892,144.569,433.116,175.735,19.455,152.980
C01361=1089.898,144.818,433.096,175.737,19.455,152.980
C01362=1089.903,145.067,433.075,175.740,19.457,152.980
C01363=1089.909,145.316,433.055,175.742,19.458,152.980
C01364=1089.915,145.565,433.034,175.745,19.459,152.980
C01365=1089.920,145.814,433.013,175.747,19.461,152.980
C01366=1089.926,146.063,432.993,175.749,19.461,152.979
C01367=1089.932,146.312,432.972,175.752,19.463,152.979
C01368=1089.937,146.562,432.952,175.755,19.464,152.979
C01369=1089.943,146.811,432.932,175.757,19.466,152.979
C01370=1089.949,147.060,432.911,175.760,19.467,152.979
C01371=1089.954,147.309,432.890,175.762,19.468,152.978
C01372=1089.959,147.558,432.869,175.764,19.469,152.978
C01373=1089.965,147.807,432.849,175.767,19.470,152.978
C01374=1089.971,148.056,432.828,175.770,19.471,152.978
C01375=1089.977,148.306,432.808,175.772,19.473,152.978
C01376=1089.982,148.555,432.787,175.774,19.473,152.977
C01377=1089.987,148.803,432.766,175.777,19.475,152.977
C01378=1089.994,149.053,432.746,175.780,19.476,152.977
C01379=1089.999,149.302,432.725,175.782,19.477,152.977
C01380=1090.004,149.551,432.705,175.785,19.478,152.977
C01381=1090.010,149.799,432.683,175.787,19.480,152.977
C01382=1090.015,150.049,432.663,175.789,19.481,152.976
C01383=1090.021,150.298,432.642,175.792,19.482,152.976
C01384=1090.026,150.548,432.621,175.795,19.483,152.976
C01385=1090.033,150.796,432.601,175.797,19.485,152.976
C01386=1090.038,151.045,432.580,175.800,19.486,152.976
C01387=1090.044,151.295,432.559,175.802,19.487,152.975
C01388=1090.049,151.543,432.538,175.804,19.488,152.975
C01389=1090.055,151.792,432.517,175.807,19.489,152.975
C01390=1090.060,152.041,432.497,175.810,19.490,152.975
C01391=1090.066,152.291,432.475,175.812,19.491,152.975
C01392=1090.071,152.540,432.455,175.815,19.493,152.974
C01393=1090.077,152.789,432.434,175.818,19.494,152.974
C01394=1090.082,153.037,432.413,175.819,19.495,152.974
C01395=1090.088,153.287,432.392,175.822,19.496,152.974
C01396=1090.094,153.536,432.371,175.825,19.498,152.974
C01397=1090.099,153.785,432.350,175.828,19.499,152.973
C01398=1090.105,154.034,432.330,175.830,19.500,152.973
C01399=1090.111,154.283,432.308,175.833,19.501,152.973
C01400=1090.116,154.532,432.288,175.835,19.502,152.973
C01401=1090.122,154.781,432.266,175.837,19.503,152.973
C01402=1090.128,155.030,432.246,175.840,19.504,152.972
C01403=1090.133,155.279,432.224,175.843,19.505,152.972
C01404=1090.139,155.529,432.203,175.845,19.507,152.972
C01405=1090.145,155.777,432.182,175.848,19.508,152.972
C01406=1090.150,156.026,432.162,175.851,19.509,152.972
C01407=1090.156,156.275,432.140,175.853,19.510,152.971
C01408=1090.161,156.525,432.119,175.855,19.511,152.971
C01409=1090.166,156.773,432.098,175.858,19.513,152.971
C01410=1090.172,157.023,432.077,175.861,19.514,152.971
C01411=1090.178,157.272,432.055,175.863,19.515,152.971
C01412=1090.183,157.520,432.034,175.866,19.516,152.970
C01413=1090.189,157.770,432.013,175.869,19.517,152.970
C01414=1090.195,158.019,431.992,175.871,19.518,152.970
C01415=1090.200,158.268,431.971,175.873,19.519,152.970
C01416=1090.206,158.517,431.950,175.876,19.520,152.970
C01417=1090.212,158.765,431.928,175.879,19.522,152.969
C01418=1090.217,159.015,431.908,175.881,19.523,152.969
C01419=1090.222,159.264,431.886,175.884,19.524,152.969
C01420=1090.229,159.541,431.862,175.887,19.525,152.969
C01421=1090.235,159.818,431.839,175.889,19.527,152.969
C01422=1090.242,160.095,431.815,175.892,19.528,152.968
C01423=1090.248,160.372,431.791,175.896,19.529,152.968
C01424=1090.253,160.622,431.770,175.898,19.530,152.968
C01425=1090.258,160.870,431.749,175.900,19.531,152.968
C01426=1090.264,161.120,431.727,175.903,19.532,152.967
C01427=1090.270,161.369,431.707,175.906,19.533,152.967
C01428=1090.276,161.618,431.685,175.909,19.535,152.967
C01429=1090.281,161.867,431.663,175.911,19.536,152.967
C01430=1090.286,162.115,431.642,175.914,19.537,152.966
C01431=1090.292,162.365,431.621,175.917,19.538,152.966
C01432=1090.297,162.614,431.599,175.918,19.539,152.966
C01433=1090.302,162.862,431.578,175.921,19.540,152.966
C01434=1090.308,163.112,431.556,175.924,19.542,152.966
C01435=1090.313,163.360,431.534,175.926,19.543,152.966
C01436=1090.319,163.610,431.513,175.929,19.544,152.965
C01437=1090.324,163.859,431.492,175.932,19.545,152.965
C01438=1090.330,164.108,431.470,175.934,19.546,152.965
C01439=1090.335,164.357,431.448,175.937,19.548,152.965
C01440=1090.341,164.606,431.427,175.940,19.549,152.964
C01441=1090.347,164.855,431.405,175.943,19.550,152.964
C01442=1090.352,165.104,431.383,175.945,19.551,152.964
C01443=1090.357,165.353,431.363,175.947,19.552,152.964
C01444=1090.362,165.602,431.341,175.950,19.553,152.964
C01445=1090.368,165.851,431.319,175.953,19.554,152.963
C01446=1090.373,166.100,431.297,175.955,19.556,152.963
C01447=1090.379,166.349,431.276,175.958,19.557,152.963
C01448=1090.385,166.598,431.254,175.961,19.558,152.963
C01449=1090.390,166.847,431.232,175.963,19.559,152.962
C01450=1090.396,167.096,431.211,175.966,19.561,152.962
C01451=1090.401,167.345,431.189,175.969,19.562,152.962
C01452=1090.406,167.593,431.167,175.972,19.563,152.962
C01453=1090.412,167.843,431.145,175.974,19.564,152.962
C01454=1090.417,168.091,431.124,175.977,19.565,152.961
C01455=1090.423,168.341,431.102,175.979,19.566,152.961
C01456=1090.428,168.589,431.080,175.982,19.567,152.961
C01457=1090.434,168.839,431.058,175.984,19.568,152.961
C01458=1090.439,169.087,431.037,175.987,19.569,152.961
C01459=1090.445,169.337,431.015,175.990,19.570,152.960
C01460=1090.450,169.585,430.993,175.992,19.572,152.960
C01461=1090.456,169.835,430.971,175.995,19.573,152.960
C01462=1090.462,170.084,430.950,175.998,19.574,152.960
C01463=1090.467,170.333,430.928,176.000,19.575,152.959
C01464=1090.473,170.582,430.906,176.003,19.576,152.959
C01465=1090.478,170.830,430.884,176.006,19.577,152.959
C01466=1090.484,171.080,430.862,176.009,19.578,152.959
C01467=1090.489,171.328,430.840,176.012,19.579,152.958
C01468=1090.495,171.578,430.818,176.014,19.580,152.958
C01469=1090.500,171.826,430.797,176.016,19.581,152.958
C01470=1090.505,172.076,430.774,176.019,19.583,152.958
C01471=1090.512,172.324,430.752,176.022,19.584,152.958
C01472=1090.517,172.573,430.730,176.024,19.585,152.957
C01473=1090.523,172.822,430.708,176.027,19.586,152.957
C01474=1090.528,173.071,430.687,176.030,19.587,152.957
C01475=1090.534,173.320,430.665,176.033,19.588,152.957
C01476=1090.540,173.569,430.642,176.035,19.589,152.956
C01477=1090.544,173.818,430.620,176.038,19.590,152.956
C01478=1090.551,174.067,430.599,176.041,19.591,152.956
C01479=1090.556,174.317,430.576,176.043,19.592,152.956
C01480=1090.562,174.565,430.554,176.046,19.594,152.955
C01481=1090.567,174.814,430.532,176.049,19.595,152.955
C01482=1090.572,175.063,430.510,176.052,19.596,152.955
C01483=1090.579,175.312,430.488,176.055,19.597,152.955
C01484=1090.584,175.589,430.463,176.057,19.598,152.954
C01485=1090.591,175.866,430.439,176.060,19.599,152.954
C01486=1090.597,176.142,430.415,176.064,19.600,152.954
C01487=1090.603,176.419,430.390,176.066,19.601,152.954
C01488=1090.609,176.668,430.368,176.069,19.602,152.953
C01489=1090.615,176.917,430.345,176.072,19.604,152.953
C01490=1090.620,177.166,430.323,176.075,19.605,152.953
C01491=1090.626,177.415,430.301,176.078,19.606,152.953
C01492=1090.632,177.664,430.278,176.080,19.607,152.952
C01493=1090.637,177.913,430.257,176.083,19.608,152.952
C01494=1090.643,178.162,430.234,176.086,19.609,152.952
C01495=1090.648,178.411,430.212,176.089,19.610,152.952
C01496=1090.654,178.660,430.189,176.091,19.611,152.951
C01497=1090.660,178.909,430.168,176.094,19.612,152.951
C01498=1090.665,179.157,430.145,176.097,19.613,152.951
C01499=1090.671,179.407,430.123,176.100,19.614,152.950
C01500=1090.677,179.656,430.100,176.103,19.615,152.950
C01501=1090.682,179.904,430.078,176.106,19.616,152.950
C01502=1090.688,180.153,430.055,176.108,19.617,152.950
C01503=1090.694,180.402,430.034,176.111,19.618,152.949
C01504=1090.700,180.651,430.011,176.114,19.619,152.949
C01505=1090.705,180.901,429.989,176.117,19.620,152.949
C01506=1090.710,181.149,429.966,176.119,19.621,152.949
C01507=1090.717,181.398,429.944,176.122,19.622,152.948
C01508=1090.722,181.647,429.922,176.125,19.623,152.948
C01509=1090.728,181.896,429.899,176.128,19.624,152.948
C01510=1090.734,182.145,429.877,176.131,19.625,152.947
C01511=1090.739,182.393,429.854,176.133,19.626,152.947
C01512=1090.745,182.642,429.831,176.136,19.627,152.947
C01513=1090.750,182.892,429.809,176.139,19.628,152.947
C01514=1090.757,183.140,429.787,176.142,19.629,152.946
C01515=1090.763,183.389,429.764,176.145,19.630,152.946
C01516=1090.768,183.639,429.742,176.148,19.631,152.946
C01517=1090.773,183.887,429.719,176.150,19.632,152.945
C01518=1090.780,184.136,429.697,176.153,19.633,152.945
C01519=1090.785,184.385,429.674,176.156,19.634,152.945
C01520=1090.791,184.634,429.652,176.159,19.635,152.945
C01521=1090.797,184.883,429.629,176.161,19.636,152.944
C01522=1090.803,185.132,429.606,176.164,19.636,152.944
C01523=1090.808,185.381,429.583,176.167,19.638,152.944
C01524=1090.813,185.630,429.561,176.170,19.639,152.944
C01525=1090.819,185.878,429.538,176.173,19.640,152.943
C01526=1090.824,186.127,429.515,176.175,19.641,152.943
C01527=1090.830,186.377,429.493,176.178,19.642,152.943
C01528=1090.835,186.625,429.470,176.181,19.643,152.943
C01529=1090.841,186.874,429.447,176.184,19.644,152.942
C01530=1090.846,187.123,429.424,176.186,19.645,152.942
C01531=1090.852,187.372,429.401,176.189,19.646,152.942
C01532=1090.858,187.621,429.378,176.192,19.647,152.941
C01533=1090.862,187.870,429.356,176.195,19.648,152.941
C01534=1090.868,188.119,429.333,176.198,19.649,152.941
C01535=1090.873,188.368,429.310,176.200,19.650,152.941
C01536=1090.879,188.616,429.287,176.203,19.651,152.940
C01537=1090.885,188.865,429.264,176.206,19.652,152.940
C01538=1090.890,189.114,429.241,176.209,19.653,152.940
C01539=1090.896,189.362,429.219,176.212,19.654,152.940
C01540=1090.901,189.612,429.195,176.214,19.656,152.939
C01541=1090.906,189.861,429.172,176.217,19.657,152.939
C01542=1090.912,190.109,429.149,176.221,19.658,152.939
C01543=1090.918,190.358,429.126,176.223,19.659,152.939
C01544=1090.924,190.607,429.103,176.226,19.660,152.938
C01545=1090.929,190.856,429.080,176.229,19.661,152.938
C01546=1090.934,191.105,429.057,176.232,19.662,152.938
C01547=1090.939,191.354,429.034,176.235,19.663,152.938
C01548=1090.945,191.631,429.009,176.238,19.664,152.937
C01549=1090.952,191.907,428.983,176.241,19.666,152.937
C01550=1090.958,192.183,428.957,176.244,19.667,152.937
C01551=1090.964,192.460,428.931,176.247,19.668,152.936
C01552=1090.970,192.709,428.909,176.251,19.669,152.936
C01553=1090.976,192.958,428.886,176.253,19.670,152.936
C01554=1090.981,193.206,428.863,176.256,19.671,152.936
C01555=1090.986,193.456,428.839,176.259,19.672,152.935
C01556=1090.992,193.705,428.816,176.262,19.673,152.935
C01557=1090.997,193.953,428.794,176.264,19.674,152.935
C01558=1091.003,194.202,428.771,176.267,19.675,152.934
C01559=1091.008,194.451,428.747,176.270,19.676,152.934
C01560=1091.014,194.699,428.723,176.273,19.677,152.934
C01561=1091.020,194.948,428.700,176.276,19.678,152.934
C01562=1091.026,195.197,428.678,176.278,19.679,152.933
C01563=1091.031,195.446,428.654,176.281,19.680,152.933
C01564=1091.036,195.695,428.631,176.285,19.681,152.933
C01565=1091.042,195.943,428.607,176.288,19.682,152.932
C01566=1091.048,196.192,428.584,176.291,19.683,152.932
C01567=1091.053,196.441,428.561,176.293,19.684,152.932
C01568=1091.059,196.690,428.538,176.296,19.685,152.932
C01569=1091.065,196.939,428.514,176.299,19.686,152.931
C01570=1091.071,197.188,428.491,176.302,19.687,152.931
C01571=1091.076,197.437,428.467,176.305,19.688,152.931
C01572=1091.082,197.686,428.444,176.308,19.689,152.931
C01573=1091.088,197.935,428.421,176.311,19.690,152.930
C01574=1091.093,198.184,428.397,176.313,19.691,152.930
C01575=1091.099,198.433,428.374,176.317,19.692,152.930
C01576=1091.105,198.681,428.351,176.320,19.693,152.929
C01577=1091.110,198.930,428.327,176.323,19.694,152.929
C01578=1091.115,199.179,428.304,176.325,19.695,152.929
C01579=1091.121,199.427,428.281,176.328,19.696,152.928
C01580=1091.126,199.677,428.257,176.331,19.697,152.928
C01581=1091.132,199.925,428.233,176.334,19.698,152.928
C01582=1091.138,200.174,428.210,176.337,19.699,152.928
C01583=1091.144,200.424,428.186,176.340,19.699,152.927
C01584=1091.150,200.672,428.163,176.343,19.701,152.927
C01585=1091.156,200.921,428.140,176.346,19.702,152.927
C01586=1091.161,201.169,428.116,176.349,19.703,152.926
C01587=1091.167,201.418,428.093,176.352,19.704,152.926
C01588=1091.172,201.667,428.068,176.355,19.705,152.926
C01589=1091.178,201.916,428.045,176.357,19.706,152.926
C01590=1091.184,202.165,428.021,176.360,19.707,152.925
C01591=1091.189,202.414,427.998,176.363,19.708,152.925
C01592=1091.195,202.662,427.974,176.367,19.709,152.924
C01593=1091.200,202.911,427.951,176.370,19.710,152.924
C01594=1091.206,203.160,427.927,176.373,19.711,152.924
C01595=1091.211,203.409,427.903,176.375,19.712,152.924
C01596=1091.217,203.657,427.880,176.378,19.713,152.923
C01597=1091.223,203.907,427.855,176.381,19.714,152.923
C01598=1091.228,204.156,427.832,176.384,19.715,152.923
C01599=1091.234,204.404,427.808,176.388,19.716,152.923
C01600=1091.239,204.653,427.784,176.390,19.717,152.922
C01601=1091.245,204.901,427.761,176.393,19.718,152.922
C01602=1091.251,205.150,427.737,176.396,19.719,152.922
C01603=1091.256,205.399,427.713,176.399,19.720,152.921
C01604=1091.262,205.648,427.689,176.402,19.721,152.921
C01605=1091.268,205.897,427.665,176.405,19.722,152.921
C01606=1091.273,206.146,427.642,176.408,19.723,152.920
C01607=1091.279,206.394,427.618,176.411,19.724,152.920
C01608=1091.284,206.643,427.593,176.414,19.725,152.920
C01609=1091.290,206.892,427.570,176.417,19.726,152.920
C01610=1091.295,207.141,427.546,176.420,19.727,152.919
C01611=1091.301,207.390,427.521,176.423,19.728,152.919
C01612=1091.324,208.410,427.424,176.487,19.759,152.915
C01613=1091.332,208.789,427.387,176.491,19.762,152.914
C01614=1091.341,209.168,427.349,176.495,19.765,152.914
C01615=1091.350,209.547,427.313,176.501,19.768,152.914
C01616=1091.358,209.925,427.275,176.505,19.771,152.914
C01617=1091.364,210.174,427.250,176.507,19.772,152.914
C01618=1091.370,210.423,427.227,176.510,19.774,152.914
C01619=1091.376,210.672,427.202,176.513,19.777,152.914
C01620=1091.381,210.920,427.178,176.516,19.779,152.914
C01621=1091.386,211.169,427.154,176.519,19.780,152.914
C01622=1091.392,211.418,427.129,176.522,19.782,152.914
C01623=1091.397,211.667,427.105,176.524,19.784,152.914
C01624=1091.403,211.915,427.080,176.528,19.786,152.914
C01625=1091.409,212.164,427.055,176.530,19.788,152.913
C01626=1091.414,212.413,427.031,176.533,19.790,152.913
C01627=1091.420,212.662,427.006,176.536,19.792,152.913
C01628=1091.425,212.911,426.982,176.538,19.793,152.913
C01629=1091.431,213.159,426.957,176.542,19.796,152.913
C01630=1091.437,213.408,426.932,176.544,19.798,152.913
C01631=1091.442,213.656,426.908,176.547,19.800,152.913
C01632=1091.448,213.906,426.883,176.550,19.801,152.913
C01633=1091.454,214.154,426.858,176.553,19.804,152.913
C01634=1091.459,214.402,426.834,176.556,19.805,152.913
C01635=1091.465,214.652,426.810,176.559,19.807,152.913
C01636=1091.470,214.900,426.784,176.561,19.809,152.913
C01637=1091.476,215.149,426.759,176.565,19.811,152.913
C01638=1091.481,215.398,426.735,176.567,19.813,152.912
C01639=1091.487,215.646,426.710,176.570,19.816,152.913
C01640=1091.492,215.895,426.686,176.573,19.817,152.912
C01641=1091.498,216.144,426.661,176.576,19.819,152.912
C01642=1091.504,216.392,426.636,176.579,19.821,152.912
C01643=1091.509,216.641,426.611,176.582,19.823,152.912
C01644=1091.514,216.890,426.587,176.585,19.825,152.912
C01645=1091.520,217.138,426.562,176.588,19.827,152.912
C01646=1091.526,217.388,426.537,176.590,19.829,152.912
C01647=1091.532,217.636,426.512,176.594,19.831,152.912
C01648=1091.537,217.885,426.487,176.596,19.833,152.912
C01649=1091.542,218.133,426.462,176.599,19.835,152.912
C01650=1091.548,218.383,426.437,176.602,19.837,152.912
C01651=1091.554,218.630,426.412,176.605,19.839,152.912
C01652=1091.560,218.880,426.388,176.607,19.841,152.912
C01653=1091.566,219.128,426.362,176.611,19.843,152.911
C01654=1091.570,219.377,426.337,176.613,19.844,152.911
C01655=1091.577,219.626,426.312,176.617,19.846,152.911
C01656=1091.582,219.875,426.288,176.619,19.848,152.911
C01657=1091.588,220.123,426.262,176.622,19.850,152.911
C01658=1091.594,220.371,426.237,176.625,19.852,152.911
C01659=1091.599,220.621,426.212,176.628,19.854,152.911
C01660=1091.605,220.869,426.187,176.631,19.856,152.911
C01661=1091.610,221.118,426.163,176.634,19.858,152.911
C01662=1091.617,221.367,426.137,176.637,19.860,152.911
C01663=1091.622,221.615,426.112,176.640,19.862,152.911
C01664=1091.627,221.864,426.087,176.642,19.864,152.911
C01665=1091.636,222.247,426.049,176.647,19.867,152.910
C01666=1091.645,222.629,426.009,176.651,19.870,152.910
C01667=1091.653,223.012,425.970,176.656,19.873,152.910
C01668=1091.662,223.395,425.932,176.660,19.876,152.910
C01669=1091.667,223.644,425.906,176.663,19.878,152.910
C01670=1091.673,223.892,425.881,176.666,19.880,152.910
C01671=1091.679,224.141,425.856,176.669,19.882,152.910
C01672=1091.684,224.390,425.831,176.672,19.884,152.910
C01673=1091.690,224.638,425.806,176.675,19.886,152.910
C01674=1091.695,224.887,425.780,176.678,19.888,152.910
C01675=1091.701,225.135,425.755,176.681,19.890,152.910
C01676=1091.707,225.384,425.729,176.683,19.892,152.910
C01677=1091.712,225.633,425.704,176.687,19.894,152.910
C01678=1091.717,225.882,425.679,176.689,19.896,152.910
C01679=1091.723,226.130,425.653,176.692,19.898,152.910
C01680=1091.729,226.379,425.627,176.695,19.900,152.909
C01681=1091.735,226.627,425.602,176.698,19.902,152.909
C01682=1091.740,226.876,425.576,176.701,19.904,152.909
C01683=1091.746,227.125,425.551,176.704,19.906,152.909
C01684=1091.751,227.373,425.526,176.707,19.908,152.909
C01685=1091.757,227.622,425.500,176.710,19.910,152.909
C01686=1091.763,227.871,425.474,176.713,19.912,152.909
C01687=1091.768,228.119,425.449,176.716,19.914,152.909
C01688=1091.774,228.368,425.423,176.719,19.916,152.909
C01689=1091.780,228.617,425.398,176.721,19.918,152.909
C01690=1091.786,228.866,425.372,176.725,19.920,152.909
C01691=1091.791,229.113,425.347,176.728,19.922,152.909
C01692=1091.797,229.362,425.321,176.730,19.924,152.909
C01693=1091.803,229.611,425.296,176.734,19.926,152.909
C01694=1091.808,229.860,425.270,176.736,19.928,152.909
C01695=1091.813,230.108,425.244,176.739,19.930,152.909
C01696=1091.819,230.357,425.219,176.742,19.932,152.908
C01697=1091.825,230.606,425.193,176.745,19.934,152.908
C01698=1091.831,230.855,425.168,176.748,19.936,152.908
C01699=1091.836,231.103,425.142,176.751,19.938,152.908
C01700=1091.841,231.352,425.116,176.754,19.940,152.908
C01701=1091.847,231.601,425.090,176.757,19.942,152.908
C01702=1091.853,231.849,425.064,176.760,19.944,152.908
C01703=1091.858,232.097,425.039,176.762,19.946,152.908
C01704=1091.864,232.346,425.013,176.766,19.948,152.908
C01705=1091.870,232.595,424.987,176.769,19.951,152.908
C01706=1091.875,232.844,424.962,176.771,19.952,152.908
C01707=1091.881,233.092,424.935,176.775,19.954,152.908
C01708=1091.886,233.341,424.909,176.777,19.956,152.908
C01709=1091.892,233.589,424.884,176.780,19.958,152.908
C01710=1091.898,233.838,424.858,176.784,19.960,152.908
C01711=1091.903,234.087,424.831,176.786,19.962,152.908
C01712=1091.909,234.336,424.805,176.790,19.964,152.907
C01713=1091.914,234.585,424.780,176.792,19.966,152.908
C01714=1091.920,234.832,424.754,176.795,19.968,152.907
C01715=1091.926,235.081,424.728,176.798,19.971,152.907
C01716=1091.931,235.330,424.702,176.801,19.973,152.907
C01717=1091.940,235.704,424.663,176.806,19.976,152.907
C01718=1091.947,236.078,424.623,176.810,19.979,152.907
C01719=1091.956,236.452,424.584,176.815,19.982,152.907
C01720=1091.965,236.826,424.545,176.819,19.985,152.907
C01721=1091.971,237.075,424.519,176.822,19.987,152.907
C01722=1091.976,237.324,424.492,176.825,19.989,152.907
C01723=1091.981,237.572,424.467,176.828,19.992,152.907
C01724=1091.987,237.820,424.440,176.830,19.993,152.907
C01725=1091.992,238.069,424.414,176.834,19.995,152.907
C01726=1091.999,238.317,424.388,176.837,19.998,152.907
C01727=1092.004,238.566,424.362,176.839,19.999,152.907
C01728=1092.010,238.815,424.335,176.843,20.002,152.907
C01729=1092.016,239.064,424.309,176.846,20.004,152.907
C01730=1092.021,239.312,424.283,176.849,20.005,152.906
C01731=1092.027,239.561,424.257,176.852,20.008,152.906
C01732=1092.033,239.809,424.230,176.855,20.010,152.906
C01733=1092.038,240.058,424.204,176.857,20.012,152.906
C01734=1092.044,240.307,424.178,176.861,20.014,152.906
C01735=1092.050,240.555,424.151,176.863,20.016,152.906
C01736=1092.055,240.804,424.125,176.866,20.018,152.906
C01737=1092.061,241.052,424.098,176.870,20.020,152.906
C01738=1092.067,241.301,424.072,176.872,20.022,152.906
C01739=1092.072,241.549,424.046,176.876,20.024,152.906
C01740=1092.077,241.797,424.019,176.879,20.026,152.906
C01741=1092.083,242.046,423.993,176.881,20.028,152.906
C01742=1092.089,242.295,423.967,176.885,20.030,152.906
C01743=1092.094,242.543,423.940,176.888,20.033,152.906
C01744=1092.100,242.791,423.914,176.890,20.035,152.906
C01745=1092.106,243.040,423.887,176.894,20.037,152.906
C01746=1092.112,243.289,423.861,176.897,20.039,152.906
C01747=1092.118,243.538,423.834,176.899,20.041,152.906
C01748=1092.122,243.786,423.807,176.902,20.043,152.906
C01749=1092.128,244.034,423.780,176.906,20.045,152.905
C01750=1092.133,244.283,423.755,176.908,20.047,152.906
C01751=1092.139,244.531,423.728,176.912,20.049,152.905
C01752=1092.145,244.780,423.701,176.915,20.052,152.905
C01753=1092.151,245.029,423.674,176.917,20.053,152.905
C01754=1092.156,245.278,423.647,176.920,20.056,152.905
C01755=1092.162,245.526,423.620,176.924,20.058,152.905
C01756=1092.168,245.774,423.594,176.926,20.060,152.905
C01757=1092.173,246.023,423.568,176.929,20.062,152.905
C01758=1092.178,246.272,423.541,176.933,20.065,152.905
C01759=1092.184,246.520,423.514,176.935,20.066,152.905
C01760=1092.190,246.769,423.487,176.938,20.069,152.905
C01761=1092.196,247.017,423.461,176.942,20.071,152.905
C01762=1092.201,247.266,423.433,176.944,20.073,152.905
C01763=1092.207,247.514,423.407,176.947,20.075,152.905
C01764=1092.212,247.762,423.380,176.951,20.077,152.905
C01765=1092.217,248.011,423.353,176.953,20.079,152.905
C01766=1092.223,248.259,423.326,176.956,20.082,152.905
C01767=1092.228,248.508,423.299,176.959,20.084,152.905
C01768=1092.234,248.756,423.272,176.963,20.086,152.905
C01769=1092.242,249.124,423.232,176.967,20.089,152.905
C01770=1092.251,249.491,423.193,176.971,20.092,152.905
C01771=1092.259,249.858,423.152,176.976,20.096,152.905
C01772=1092.267,250.225,423.112,176.980,20.099,152.905
C01773=1092.272,250.474,423.085,176.983,20.101,152.905
C01774=1092.278,250.722,423.059,176.986,20.103,152.905
C01775=1092.283,250.971,423.031,176.989,20.106,152.905
C01776=1092.289,251.219,423.005,176.992,20.108,152.905
C01777=1092.294,251.467,422.977,176.995,20.110,152.905
C01778=1092.301,251.716,422.950,176.998,20.112,152.905
C01779=1092.306,251.965,422.923,177.001,20.114,152.905
C01780=1092.312,252.213,422.896,177.004,20.117,152.905
C01781=1092.317,252.462,422.869,177.007,20.119,152.905
C01782=1092.323,252.710,422.841,177.010,20.121,152.905
C01783=1092.328,252.958,422.814,177.013,20.123,152.904
C01784=1092.334,253.207,422.787,177.016,20.125,152.905
C01785=1092.339,253.456,422.759,177.019,20.127,152.904
C01786=1092.345,253.704,422.732,177.023,20.130,152.904
C01787=1092.350,253.953,422.705,177.025,20.132,152.904
C01788=1092.356,254.200,422.678,177.028,20.134,152.904
C01789=1092.361,254.449,422.651,177.031,20.137,152.904
C01790=1092.368,254.698,422.624,177.034,20.138,152.904
C01791=1092.373,254.946,422.596,177.037,20.141,152.904
C01792=1092.378,255.195,422.568,177.040,20.143,152.904
C01793=1092.384,255.443,422.542,177.044,20.145,152.904
C01794=1092.390,255.692,422.513,177.046,20.147,152.904
C01795=1092.396,255.940,422.487,177.049,20.149,152.904
C01796=1092.401,256.188,422.459,177.053,20.152,152.904
C01797=1092.407,256.437,422.432,177.056,20.154,152.904
C01798=1092.413,256.685,422.404,177.058,20.156,152.904
C01799=1092.418,256.934,422.377,177.061,20.159,152.904
C01800=1092.424,257.182,422.349,177.065,20.161,152.904
C01801=1092.429,257.431,422.322,177.068,20.163,152.904
C01802=1092.436,257.679,422.294,177.071,20.165,152.904
C01803=1092.441,257.928,422.267,177.074,20.167,152.904
C01804=1092.446,258.176,422.239,177.077,20.169,152.904
C01805=1092.452,258.425,422.212,177.080,20.172,152.904
C01806=1092.458,258.673,422.184,177.083,20.173,152.904
C01807=1092.464,258.920,422.157,177.086,20.176,152.904
C01808=1092.469,259.170,422.129,177.089,20.178,152.904
C01809=1092.475,259.418,422.101,177.092,20.180,152.904
C01810=1092.481,259.667,422.074,177.095,20.182,152.904
C01811=1092.486,259.915,422.046,177.098,20.185,152.904
C01812=1092.492,260.163,422.018,177.101,20.187,152.904
C01813=1092.498,260.412,421.991,177.105,20.189,152.904
